// TIA Portal V17 export
// export: Created 2025-07-01T14:25:48.2523347Z, ExportSetting WithDefaults, DisplayName Totally Integrated Automation Portal, DisplayVersion V17 Update 8, DisplayName TIA Portal Openness, DisplayVersion V17 Update 8, DisplayName TIA Portal Version Control Interface, DisplayVersion V17, DisplayName SINAMICS Startdrive Advanced, DisplayVersion V17 SP2, DisplayName SINAMICS Startdrive G110M, G120, G120C, G120D, G120P, G115D, DisplayVersion V17 SP2, DisplayName SINAMICS Startdrive G130, G150, S120, S150, SINAMICS MV, S210, DisplayVersion V17 SP2, DisplayName STEP 7 Professional, DisplayVersion V17 Update 8, DisplayName SINUMERIK ONE STEP 7 Toolbox, DisplayVersion V17 Update 12, DisplayName SINUMERIK ONE PLC Basic Program Plus, DisplayVersion V17 Update 12, DisplayName SINUMERIK 840D sl STEP 7 Toolbox, DisplayVersion V17 Update 12, DisplayName STEP 7 Safety, DisplayVersion V17 Update 6, DisplayName WinCC Advanced, DisplayVersion V17 Update 8
FUNCTION "FC2103_ELECTRICAL_CABINET" : Void   // FC2103, LAD
{ S7_Optimized_Access := 'FALSE' }
AUTHOR : ETXETAR
VERSION : 1.0
// stored: AutoNumber false, IsIECCheckEnabled false, SetENOAutomatically false, UDAEnableTagReadback false
   VAR_TEMP
      PSP_ALARM_AUX : Bool;
   END_VAR
   VAR CONSTANT
      FC_NUMBER : DInt := 2103;
   END_VAR
   VAR_TEMP   // added for the SCL form of the ladder/FBD networks
      _w1 : Bool;
   END_VAR
BEGIN

REGION Network 1: INPUTS
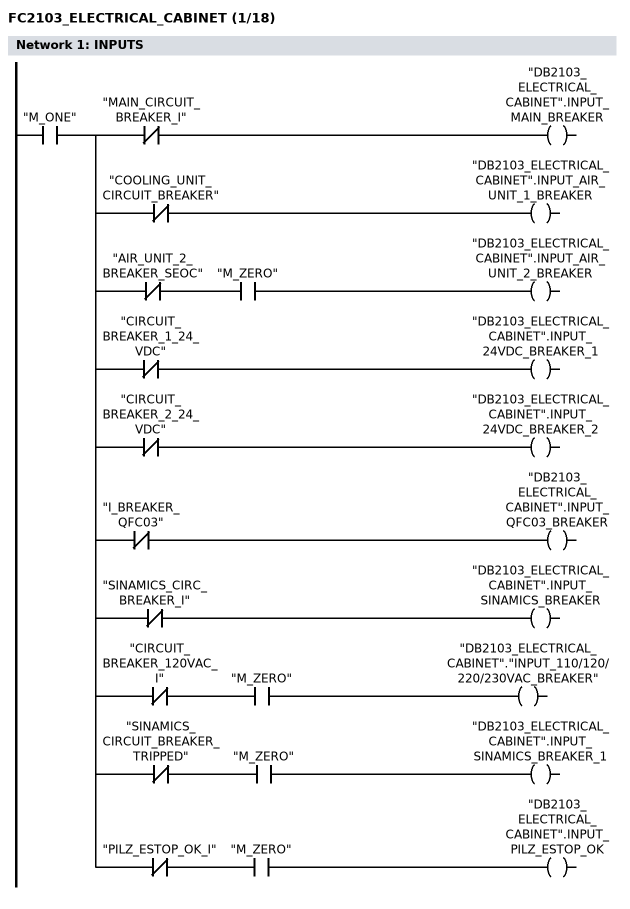
   RUNG wire#powerrail
      Contact( "M_ONE" )
      wire#w1
      I_Contact( "MAIN_CIRCUIT_BREAKER_I" )
      Coil( "DB2103_ELECTRICAL_CABINET".INPUT_MAIN_BREAKER )
   END_RUNG
   RUNG wire#w1
      I_Contact( "COOLING_UNIT_CIRCUIT_BREAKER" )
      Coil( "DB2103_ELECTRICAL_CABINET".INPUT_AIR_UNIT_1_BREAKER )
   END_RUNG
   RUNG wire#w1
      I_Contact( "AIR_UNIT_2_BREAKER_SEOC" )
      Contact( "M_ZERO" )
      Coil( "DB2103_ELECTRICAL_CABINET".INPUT_AIR_UNIT_2_BREAKER )
   END_RUNG
   RUNG wire#w1
      I_Contact( "CIRCUIT_BREAKER_1_24_VDC" )
      Coil( "DB2103_ELECTRICAL_CABINET".INPUT_24VDC_BREAKER_1 )
   END_RUNG
   RUNG wire#w1
      I_Contact( "CIRCUIT_BREAKER_2_24_VDC" )
      Coil( "DB2103_ELECTRICAL_CABINET".INPUT_24VDC_BREAKER_2 )
   END_RUNG
   RUNG wire#w1
      I_Contact( "I_BREAKER_QFC03" )
      Coil( "DB2103_ELECTRICAL_CABINET".INPUT_QFC03_BREAKER )
   END_RUNG
   RUNG wire#w1
      I_Contact( "SINAMICS_CIRC_BREAKER_I" )
      Coil( "DB2103_ELECTRICAL_CABINET".INPUT_SINAMICS_BREAKER )
   END_RUNG
   RUNG wire#w1
      I_Contact( "CIRCUIT_BREAKER_120VAC_I" )
      Contact( "M_ZERO" )
      Coil( "DB2103_ELECTRICAL_CABINET"."INPUT_110/120/220/230VAC_BREAKER" )
   END_RUNG
   RUNG wire#w1
      I_Contact( "SINAMICS_CIRCUIT_BREAKER_TRIPPED" )
      Contact( "M_ZERO" )
      Coil( "DB2103_ELECTRICAL_CABINET".INPUT_SINAMICS_BREAKER_1 )
   END_RUNG
   RUNG wire#w1
      I_Contact( "PILZ_ESTOP_OK_I" )
      Contact( "M_ZERO" )
      Coil( "DB2103_ELECTRICAL_CABINET".INPUT_PILZ_ESTOP_OK )
   END_RUNG
   // the same network as SCL:
   "DB2103_ELECTRICAL_CABINET".INPUT_MAIN_BREAKER := "M_ONE" AND NOT "MAIN_CIRCUIT_BREAKER_I";
   "DB2103_ELECTRICAL_CABINET".INPUT_AIR_UNIT_1_BREAKER := "M_ONE" AND NOT "COOLING_UNIT_CIRCUIT_BREAKER";
   "DB2103_ELECTRICAL_CABINET".INPUT_AIR_UNIT_2_BREAKER := "M_ONE" AND NOT "AIR_UNIT_2_BREAKER_SEOC" AND "M_ZERO";
   "DB2103_ELECTRICAL_CABINET".INPUT_24VDC_BREAKER_1 := "M_ONE" AND NOT "CIRCUIT_BREAKER_1_24_VDC";
   "DB2103_ELECTRICAL_CABINET".INPUT_24VDC_BREAKER_2 := "M_ONE" AND NOT "CIRCUIT_BREAKER_2_24_VDC";
   "DB2103_ELECTRICAL_CABINET".INPUT_QFC03_BREAKER := "M_ONE" AND NOT "I_BREAKER_QFC03";
   "DB2103_ELECTRICAL_CABINET".INPUT_SINAMICS_BREAKER := "M_ONE" AND NOT "SINAMICS_CIRC_BREAKER_I";
   "DB2103_ELECTRICAL_CABINET"."INPUT_110/120/220/230VAC_BREAKER" := "M_ONE" AND NOT "CIRCUIT_BREAKER_120VAC_I" AND "M_ZERO";
   "DB2103_ELECTRICAL_CABINET".INPUT_SINAMICS_BREAKER_1 := "M_ONE" AND NOT "SINAMICS_CIRCUIT_BREAKER_TRIPPED" AND "M_ZERO";
   "DB2103_ELECTRICAL_CABINET".INPUT_PILZ_ESTOP_OK := "M_ONE" AND NOT "PILZ_ESTOP_OK_I" AND "M_ZERO";
END_REGION

REGION Network 2: INPUTS
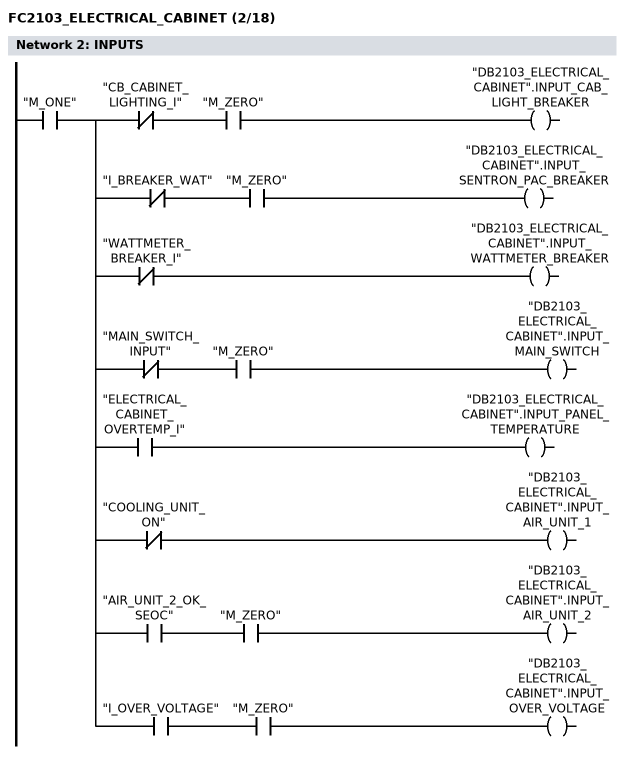
   RUNG wire#powerrail
      Contact( "M_ONE" )
      wire#w1
      I_Contact( "CB_CABINET_LIGHTING_I" )
      Contact( "M_ZERO" )
      Coil( "DB2103_ELECTRICAL_CABINET".INPUT_CAB_LIGHT_BREAKER )
   END_RUNG
   RUNG wire#w1
      I_Contact( "I_BREAKER_WAT" )
      Contact( "M_ZERO" )
      Coil( "DB2103_ELECTRICAL_CABINET".INPUT_SENTRON_PAC_BREAKER )
   END_RUNG
   RUNG wire#w1
      I_Contact( "WATTMETER_BREAKER_I" )
      Coil( "DB2103_ELECTRICAL_CABINET".INPUT_WATTMETER_BREAKER )
   END_RUNG
   RUNG wire#w1
      I_Contact( "MAIN_SWITCH_INPUT" )
      Contact( "M_ZERO" )
      Coil( "DB2103_ELECTRICAL_CABINET".INPUT_MAIN_SWITCH )
   END_RUNG
   RUNG wire#w1
      Contact( "ELECTRICAL_CABINET_OVERTEMP_I" )
      Coil( "DB2103_ELECTRICAL_CABINET".INPUT_PANEL_TEMPERATURE )
   END_RUNG
   RUNG wire#w1
      I_Contact( "COOLING_UNIT_ON" )
      Coil( "DB2103_ELECTRICAL_CABINET".INPUT_AIR_UNIT_1 )
   END_RUNG
   RUNG wire#w1
      Contact( "AIR_UNIT_2_OK_SEOC" )
      Contact( "M_ZERO" )
      Coil( "DB2103_ELECTRICAL_CABINET".INPUT_AIR_UNIT_2 )
   END_RUNG
   RUNG wire#w1
      Contact( "I_OVER_VOLTAGE" )
      Contact( "M_ZERO" )
      Coil( "DB2103_ELECTRICAL_CABINET".INPUT_OVER_VOLTAGE )
   END_RUNG
   // the same network as SCL:
   "DB2103_ELECTRICAL_CABINET".INPUT_CAB_LIGHT_BREAKER := "M_ONE" AND NOT "CB_CABINET_LIGHTING_I" AND "M_ZERO";
   "DB2103_ELECTRICAL_CABINET".INPUT_SENTRON_PAC_BREAKER := "M_ONE" AND NOT "I_BREAKER_WAT" AND "M_ZERO";
   "DB2103_ELECTRICAL_CABINET".INPUT_WATTMETER_BREAKER := "M_ONE" AND NOT "WATTMETER_BREAKER_I";
   "DB2103_ELECTRICAL_CABINET".INPUT_MAIN_SWITCH := "M_ONE" AND NOT "MAIN_SWITCH_INPUT" AND "M_ZERO";
   "DB2103_ELECTRICAL_CABINET".INPUT_PANEL_TEMPERATURE := "M_ONE" AND "ELECTRICAL_CABINET_OVERTEMP_I";
   "DB2103_ELECTRICAL_CABINET".INPUT_AIR_UNIT_1 := "M_ONE" AND NOT "COOLING_UNIT_ON";
   "DB2103_ELECTRICAL_CABINET".INPUT_AIR_UNIT_2 := "M_ONE" AND "AIR_UNIT_2_OK_SEOC" AND "M_ZERO";
   "DB2103_ELECTRICAL_CABINET".INPUT_OVER_VOLTAGE := "M_ONE" AND "I_OVER_VOLTAGE" AND "M_ZERO";
END_REGION

REGION Network 3: INPUTS
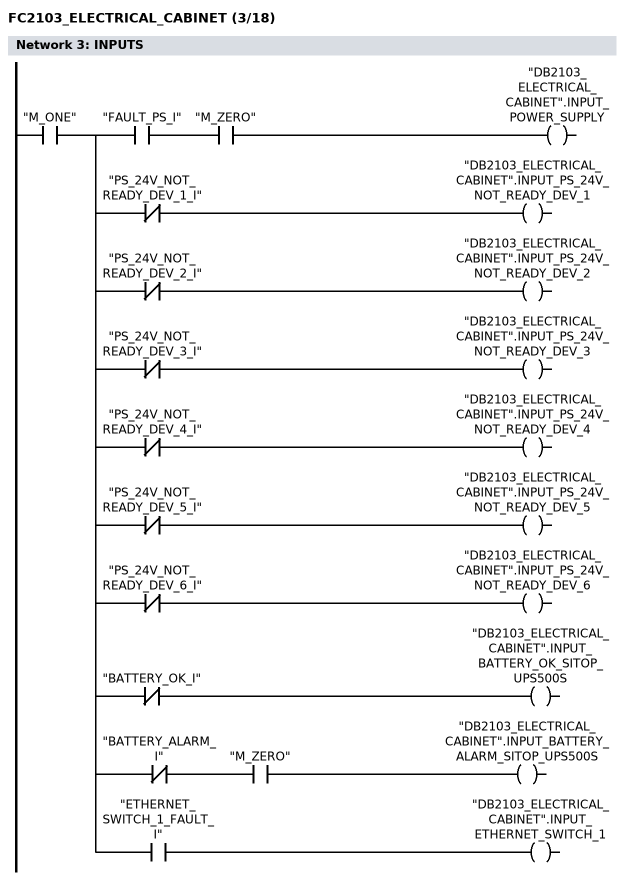
   RUNG wire#powerrail
      Contact( "M_ONE" )
      wire#w1
      Contact( "FAULT_PS_I" )
      Contact( "M_ZERO" )
      Coil( "DB2103_ELECTRICAL_CABINET".INPUT_POWER_SUPPLY )
   END_RUNG
   RUNG wire#w1
      I_Contact( "PS_24V_NOT_READY_DEV_1_I" )
      Coil( "DB2103_ELECTRICAL_CABINET".INPUT_PS_24V_NOT_READY_DEV_1 )
   END_RUNG
   RUNG wire#w1
      I_Contact( "PS_24V_NOT_READY_DEV_2_I" )
      Coil( "DB2103_ELECTRICAL_CABINET".INPUT_PS_24V_NOT_READY_DEV_2 )
   END_RUNG
   RUNG wire#w1
      I_Contact( "PS_24V_NOT_READY_DEV_3_I" )
      Coil( "DB2103_ELECTRICAL_CABINET".INPUT_PS_24V_NOT_READY_DEV_3 )
   END_RUNG
   RUNG wire#w1
      I_Contact( "PS_24V_NOT_READY_DEV_4_I" )
      Coil( "DB2103_ELECTRICAL_CABINET".INPUT_PS_24V_NOT_READY_DEV_4 )
   END_RUNG
   RUNG wire#w1
      I_Contact( "PS_24V_NOT_READY_DEV_5_I" )
      Coil( "DB2103_ELECTRICAL_CABINET".INPUT_PS_24V_NOT_READY_DEV_5 )
   END_RUNG
   RUNG wire#w1
      I_Contact( "PS_24V_NOT_READY_DEV_6_I" )
      Coil( "DB2103_ELECTRICAL_CABINET".INPUT_PS_24V_NOT_READY_DEV_6 )
   END_RUNG
   RUNG wire#w1
      I_Contact( "BATTERY_OK_I" )
      Coil( "DB2103_ELECTRICAL_CABINET".INPUT_BATTERY_OK_SITOP_UPS500S )
   END_RUNG
   RUNG wire#w1
      I_Contact( "BATTERY_ALARM_I" )
      Contact( "M_ZERO" )
      Coil( "DB2103_ELECTRICAL_CABINET".INPUT_BATTERY_ALARM_SITOP_UPS500S )
   END_RUNG
   RUNG wire#w1
      Contact( "ETHERNET_SWITCH_1_FAULT_I" )
      Coil( "DB2103_ELECTRICAL_CABINET".INPUT_ETHERNET_SWITCH_1 )
   END_RUNG
   // the same network as SCL:
   "DB2103_ELECTRICAL_CABINET".INPUT_POWER_SUPPLY := "M_ONE" AND "FAULT_PS_I" AND "M_ZERO";
   "DB2103_ELECTRICAL_CABINET".INPUT_PS_24V_NOT_READY_DEV_1 := "M_ONE" AND NOT "PS_24V_NOT_READY_DEV_1_I";
   "DB2103_ELECTRICAL_CABINET".INPUT_PS_24V_NOT_READY_DEV_2 := "M_ONE" AND NOT "PS_24V_NOT_READY_DEV_2_I";
   "DB2103_ELECTRICAL_CABINET".INPUT_PS_24V_NOT_READY_DEV_3 := "M_ONE" AND NOT "PS_24V_NOT_READY_DEV_3_I";
   "DB2103_ELECTRICAL_CABINET".INPUT_PS_24V_NOT_READY_DEV_4 := "M_ONE" AND NOT "PS_24V_NOT_READY_DEV_4_I";
   "DB2103_ELECTRICAL_CABINET".INPUT_PS_24V_NOT_READY_DEV_5 := "M_ONE" AND NOT "PS_24V_NOT_READY_DEV_5_I";
   "DB2103_ELECTRICAL_CABINET".INPUT_PS_24V_NOT_READY_DEV_6 := "M_ONE" AND NOT "PS_24V_NOT_READY_DEV_6_I";
   "DB2103_ELECTRICAL_CABINET".INPUT_BATTERY_OK_SITOP_UPS500S := "M_ONE" AND NOT "BATTERY_OK_I";
   "DB2103_ELECTRICAL_CABINET".INPUT_BATTERY_ALARM_SITOP_UPS500S := "M_ONE" AND NOT "BATTERY_ALARM_I" AND "M_ZERO";
   "DB2103_ELECTRICAL_CABINET".INPUT_ETHERNET_SWITCH_1 := "M_ONE" AND "ETHERNET_SWITCH_1_FAULT_I";
END_REGION

REGION Network 4: INPUTS
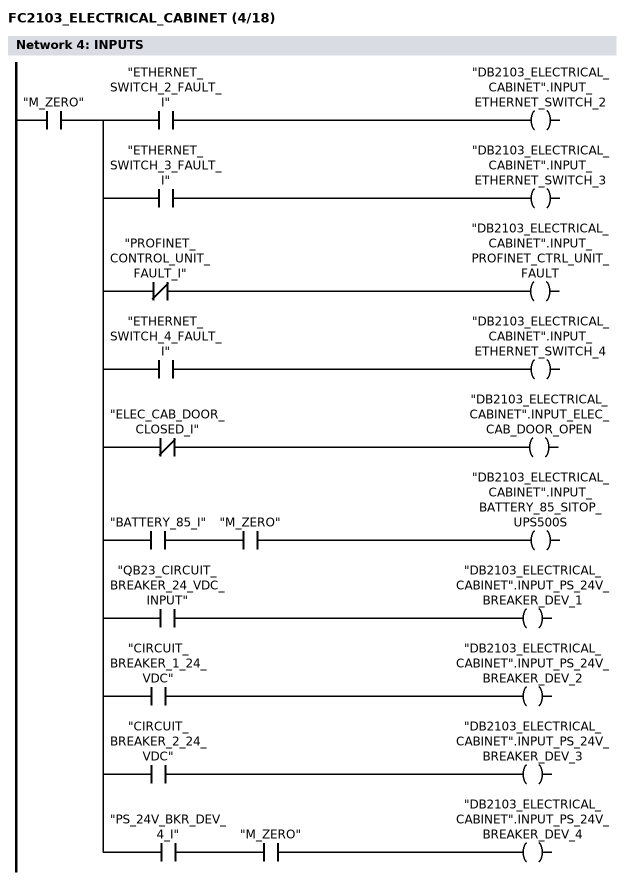
   RUNG wire#powerrail
      Contact( "M_ZERO" )
      wire#w1
      Contact( "ETHERNET_SWITCH_2_FAULT_I" )
      Coil( "DB2103_ELECTRICAL_CABINET".INPUT_ETHERNET_SWITCH_2 )
   END_RUNG
   RUNG wire#w1
      Contact( "ETHERNET_SWITCH_3_FAULT_I" )
      Coil( "DB2103_ELECTRICAL_CABINET".INPUT_ETHERNET_SWITCH_3 )
   END_RUNG
   RUNG wire#w1
      I_Contact( "PROFINET_CONTROL_UNIT_FAULT_I" )
      Coil( "DB2103_ELECTRICAL_CABINET".INPUT_PROFINET_CTRL_UNIT_FAULT )
   END_RUNG
   RUNG wire#w1
      Contact( "ETHERNET_SWITCH_4_FAULT_I" )
      Coil( "DB2103_ELECTRICAL_CABINET".INPUT_ETHERNET_SWITCH_4 )
   END_RUNG
   RUNG wire#w1
      I_Contact( "ELEC_CAB_DOOR_CLOSED_I" )
      Coil( "DB2103_ELECTRICAL_CABINET".INPUT_ELEC_CAB_DOOR_OPEN )
   END_RUNG
   RUNG wire#w1
      Contact( "BATTERY_85_I" )
      Contact( "M_ZERO" )
      Coil( "DB2103_ELECTRICAL_CABINET".INPUT_BATTERY_85_SITOP_UPS500S )
   END_RUNG
   RUNG wire#w1
      Contact( "QB23_CIRCUIT_BREAKER_24_VDC_INPUT" )
      Coil( "DB2103_ELECTRICAL_CABINET".INPUT_PS_24V_BREAKER_DEV_1 )
   END_RUNG
   RUNG wire#w1
      Contact( "CIRCUIT_BREAKER_1_24_VDC" )
      Coil( "DB2103_ELECTRICAL_CABINET".INPUT_PS_24V_BREAKER_DEV_2 )
   END_RUNG
   RUNG wire#w1
      Contact( "CIRCUIT_BREAKER_2_24_VDC" )
      Coil( "DB2103_ELECTRICAL_CABINET".INPUT_PS_24V_BREAKER_DEV_3 )
   END_RUNG
   RUNG wire#w1
      Contact( "PS_24V_BKR_DEV_4_I" )
      Contact( "M_ZERO" )
      Coil( "DB2103_ELECTRICAL_CABINET".INPUT_PS_24V_BREAKER_DEV_4 )
   END_RUNG
   // the same network as SCL:
   "DB2103_ELECTRICAL_CABINET".INPUT_ETHERNET_SWITCH_2 := "M_ZERO" AND "ETHERNET_SWITCH_2_FAULT_I";
   "DB2103_ELECTRICAL_CABINET".INPUT_ETHERNET_SWITCH_3 := "M_ZERO" AND "ETHERNET_SWITCH_3_FAULT_I";
   "DB2103_ELECTRICAL_CABINET".INPUT_PROFINET_CTRL_UNIT_FAULT := "M_ZERO" AND NOT "PROFINET_CONTROL_UNIT_FAULT_I";
   "DB2103_ELECTRICAL_CABINET".INPUT_ETHERNET_SWITCH_4 := "M_ZERO" AND "ETHERNET_SWITCH_4_FAULT_I";
   "DB2103_ELECTRICAL_CABINET".INPUT_ELEC_CAB_DOOR_OPEN := "M_ZERO" AND NOT "ELEC_CAB_DOOR_CLOSED_I";
   "DB2103_ELECTRICAL_CABINET".INPUT_BATTERY_85_SITOP_UPS500S := "M_ZERO" AND "BATTERY_85_I" AND "M_ZERO";
   "DB2103_ELECTRICAL_CABINET".INPUT_PS_24V_BREAKER_DEV_1 := "M_ZERO" AND "QB23_CIRCUIT_BREAKER_24_VDC_INPUT";
   "DB2103_ELECTRICAL_CABINET".INPUT_PS_24V_BREAKER_DEV_2 := "M_ZERO" AND "CIRCUIT_BREAKER_1_24_VDC";
   "DB2103_ELECTRICAL_CABINET".INPUT_PS_24V_BREAKER_DEV_3 := "M_ZERO" AND "CIRCUIT_BREAKER_2_24_VDC";
   "DB2103_ELECTRICAL_CABINET".INPUT_PS_24V_BREAKER_DEV_4 := "M_ZERO" AND "PS_24V_BKR_DEV_4_I" AND "M_ZERO";
END_REGION

REGION Network 5: INPUTS
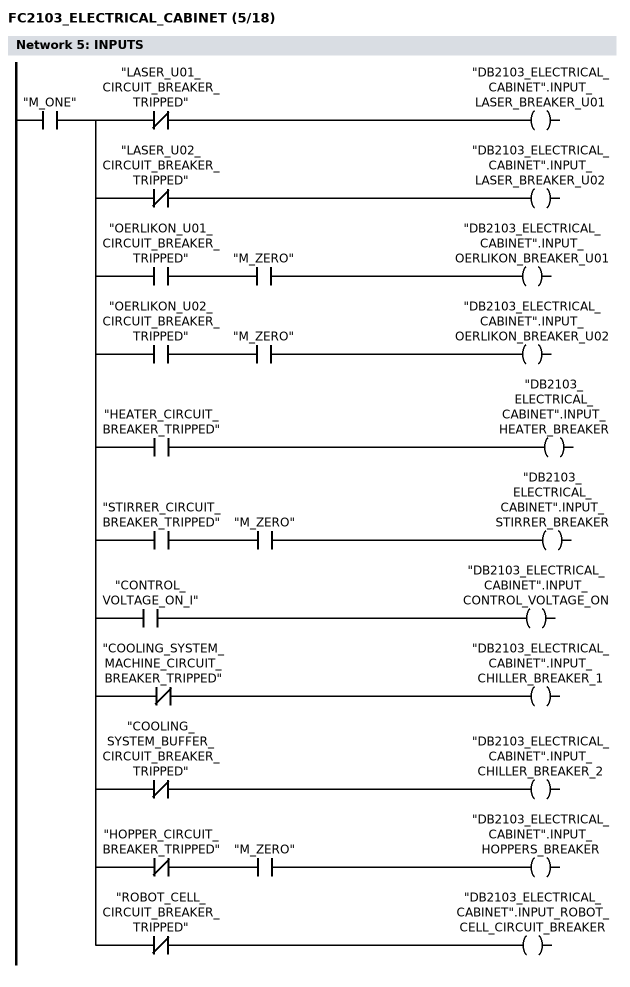
   RUNG wire#powerrail
      Contact( "M_ONE" )
      wire#w1
      I_Contact( "LASER_U01_CIRCUIT_BREAKER_TRIPPED" )
      Coil( "DB2103_ELECTRICAL_CABINET".INPUT_LASER_BREAKER_U01 )
   END_RUNG
   RUNG wire#w1
      I_Contact( "LASER_U02_CIRCUIT_BREAKER_TRIPPED" )
      Coil( "DB2103_ELECTRICAL_CABINET".INPUT_LASER_BREAKER_U02 )
   END_RUNG
   RUNG wire#w1
      Contact( "OERLIKON_U01_CIRCUIT_BREAKER_TRIPPED" )
      Contact( "M_ZERO" )
      Coil( "DB2103_ELECTRICAL_CABINET".INPUT_OERLIKON_BREAKER_U01 )
   END_RUNG
   RUNG wire#w1
      Contact( "OERLIKON_U02_CIRCUIT_BREAKER_TRIPPED" )
      Contact( "M_ZERO" )
      Coil( "DB2103_ELECTRICAL_CABINET".INPUT_OERLIKON_BREAKER_U02 )
   END_RUNG
   RUNG wire#w1
      Contact( "HEATER_CIRCUIT_BREAKER_TRIPPED" )
      Coil( "DB2103_ELECTRICAL_CABINET".INPUT_HEATER_BREAKER )
   END_RUNG
   RUNG wire#w1
      Contact( "STIRRER_CIRCUIT_BREAKER_TRIPPED" )
      Contact( "M_ZERO" )
      Coil( "DB2103_ELECTRICAL_CABINET".INPUT_STIRRER_BREAKER )
   END_RUNG
   RUNG wire#w1
      Contact( "CONTROL_VOLTAGE_ON_I" )
      Coil( "DB2103_ELECTRICAL_CABINET".INPUT_CONTROL_VOLTAGE_ON )
   END_RUNG
   RUNG wire#w1
      I_Contact( "COOLING_SYSTEM_MACHINE_CIRCUIT_BREAKER_TRIPPED" )
      Coil( "DB2103_ELECTRICAL_CABINET".INPUT_CHILLER_BREAKER_1 )
   END_RUNG
   RUNG wire#w1
      I_Contact( "COOLING_SYSTEM_BUFFER_CIRCUIT_BREAKER_TRIPPED" )
      Coil( "DB2103_ELECTRICAL_CABINET".INPUT_CHILLER_BREAKER_2 )
   END_RUNG
   RUNG wire#w1
      I_Contact( "HOPPER_CIRCUIT_BREAKER_TRIPPED" )
      Contact( "M_ZERO" )
      Coil( "DB2103_ELECTRICAL_CABINET".INPUT_HOPPERS_BREAKER )
   END_RUNG
   RUNG wire#w1
      I_Contact( "ROBOT_CELL_CIRCUIT_BREAKER_TRIPPED" )
      Coil( "DB2103_ELECTRICAL_CABINET".INPUT_ROBOT_CELL_CIRCUIT_BREAKER )
   END_RUNG
   // the same network as SCL:
   "DB2103_ELECTRICAL_CABINET".INPUT_LASER_BREAKER_U01 := "M_ONE" AND NOT "LASER_U01_CIRCUIT_BREAKER_TRIPPED";
   "DB2103_ELECTRICAL_CABINET".INPUT_LASER_BREAKER_U02 := "M_ONE" AND NOT "LASER_U02_CIRCUIT_BREAKER_TRIPPED";
   "DB2103_ELECTRICAL_CABINET".INPUT_OERLIKON_BREAKER_U01 := "M_ONE" AND "OERLIKON_U01_CIRCUIT_BREAKER_TRIPPED" AND "M_ZERO";
   "DB2103_ELECTRICAL_CABINET".INPUT_OERLIKON_BREAKER_U02 := "M_ONE" AND "OERLIKON_U02_CIRCUIT_BREAKER_TRIPPED" AND "M_ZERO";
   "DB2103_ELECTRICAL_CABINET".INPUT_HEATER_BREAKER := "M_ONE" AND "HEATER_CIRCUIT_BREAKER_TRIPPED";
   "DB2103_ELECTRICAL_CABINET".INPUT_STIRRER_BREAKER := "M_ONE" AND "STIRRER_CIRCUIT_BREAKER_TRIPPED" AND "M_ZERO";
   "DB2103_ELECTRICAL_CABINET".INPUT_CONTROL_VOLTAGE_ON := "M_ONE" AND "CONTROL_VOLTAGE_ON_I";
   "DB2103_ELECTRICAL_CABINET".INPUT_CHILLER_BREAKER_1 := "M_ONE" AND NOT "COOLING_SYSTEM_MACHINE_CIRCUIT_BREAKER_TRIPPED";
   "DB2103_ELECTRICAL_CABINET".INPUT_CHILLER_BREAKER_2 := "M_ONE" AND NOT "COOLING_SYSTEM_BUFFER_CIRCUIT_BREAKER_TRIPPED";
   "DB2103_ELECTRICAL_CABINET".INPUT_HOPPERS_BREAKER := "M_ONE" AND NOT "HOPPER_CIRCUIT_BREAKER_TRIPPED" AND "M_ZERO";
   "DB2103_ELECTRICAL_CABINET".INPUT_ROBOT_CELL_CIRCUIT_BREAKER := "M_ONE" AND NOT "ROBOT_CELL_CIRCUIT_BREAKER_TRIPPED";
END_REGION

REGION Network 6: INPUTS
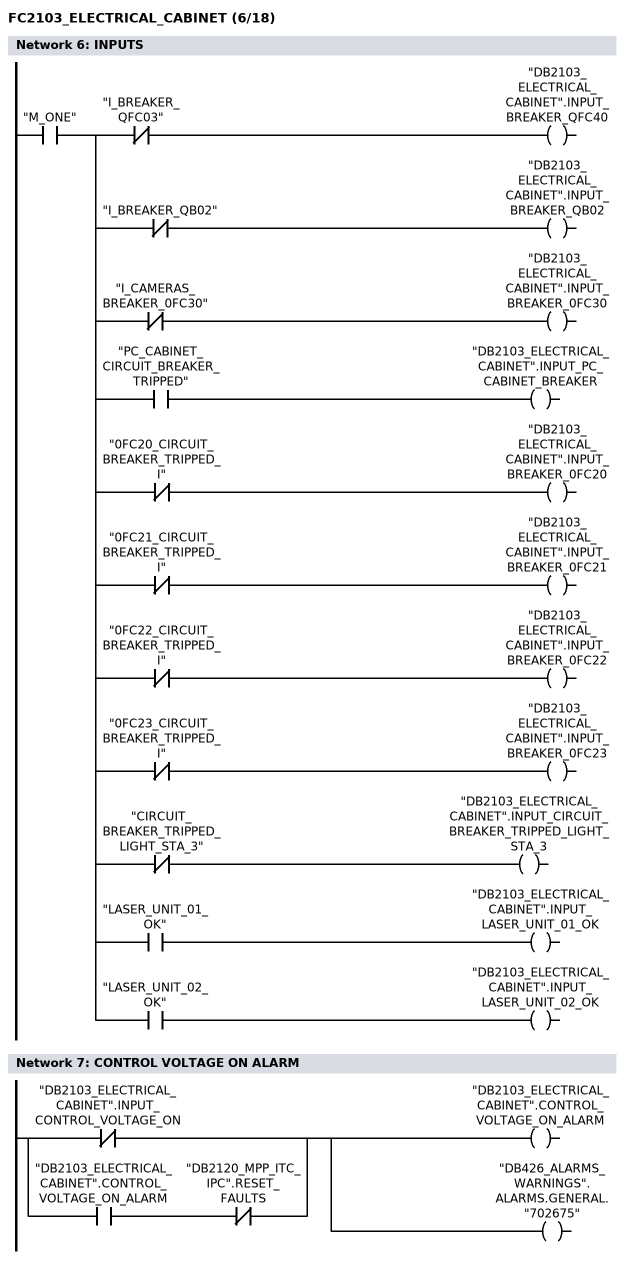
   RUNG wire#powerrail
      Contact( "M_ONE" )
      wire#w1
      I_Contact( "I_BREAKER_QFC03" )
      Coil( "DB2103_ELECTRICAL_CABINET".INPUT_BREAKER_QFC40 )
   END_RUNG
   RUNG wire#w1
      I_Contact( "I_BREAKER_QB02" )
      Coil( "DB2103_ELECTRICAL_CABINET".INPUT_BREAKER_QB02 )
   END_RUNG
   RUNG wire#w1
      I_Contact( "I_CAMERAS_BREAKER_0FC30" )
      Coil( "DB2103_ELECTRICAL_CABINET".INPUT_BREAKER_0FC30 )
   END_RUNG
   RUNG wire#w1
      Contact( "PC_CABINET_CIRCUIT_BREAKER_TRIPPED" )
      Coil( "DB2103_ELECTRICAL_CABINET".INPUT_PC_CABINET_BREAKER )
   END_RUNG
   RUNG wire#w1
      I_Contact( "0FC20_CIRCUIT_BREAKER_TRIPPED_I" )
      Coil( "DB2103_ELECTRICAL_CABINET".INPUT_BREAKER_0FC20 )
   END_RUNG
   RUNG wire#w1
      I_Contact( "0FC21_CIRCUIT_BREAKER_TRIPPED_I" )
      Coil( "DB2103_ELECTRICAL_CABINET".INPUT_BREAKER_0FC21 )
   END_RUNG
   RUNG wire#w1
      I_Contact( "0FC22_CIRCUIT_BREAKER_TRIPPED_I" )
      Coil( "DB2103_ELECTRICAL_CABINET".INPUT_BREAKER_0FC22 )
   END_RUNG
   RUNG wire#w1
      I_Contact( "0FC23_CIRCUIT_BREAKER_TRIPPED_I" )
      Coil( "DB2103_ELECTRICAL_CABINET".INPUT_BREAKER_0FC23 )
   END_RUNG
   RUNG wire#w1
      I_Contact( "CIRCUIT_BREAKER_TRIPPED_LIGHT_STA_3" )
      Coil( "DB2103_ELECTRICAL_CABINET".INPUT_CIRCUIT_BREAKER_TRIPPED_LIGHT_STA_3 )
   END_RUNG
   RUNG wire#w1
      Contact( "LASER_UNIT_01_OK" )
      Coil( "DB2103_ELECTRICAL_CABINET".INPUT_LASER_UNIT_01_OK )
   END_RUNG
   RUNG wire#w1
      Contact( "LASER_UNIT_02_OK" )
      Coil( "DB2103_ELECTRICAL_CABINET".INPUT_LASER_UNIT_02_OK )
   END_RUNG
   // the same network as SCL:
   "DB2103_ELECTRICAL_CABINET".INPUT_BREAKER_QFC40 := "M_ONE" AND NOT "I_BREAKER_QFC03";
   "DB2103_ELECTRICAL_CABINET".INPUT_BREAKER_QB02 := "M_ONE" AND NOT "I_BREAKER_QB02";
   "DB2103_ELECTRICAL_CABINET".INPUT_BREAKER_0FC30 := "M_ONE" AND NOT "I_CAMERAS_BREAKER_0FC30";
   "DB2103_ELECTRICAL_CABINET".INPUT_PC_CABINET_BREAKER := "M_ONE" AND "PC_CABINET_CIRCUIT_BREAKER_TRIPPED";
   "DB2103_ELECTRICAL_CABINET".INPUT_BREAKER_0FC20 := "M_ONE" AND NOT "0FC20_CIRCUIT_BREAKER_TRIPPED_I";
   "DB2103_ELECTRICAL_CABINET".INPUT_BREAKER_0FC21 := "M_ONE" AND NOT "0FC21_CIRCUIT_BREAKER_TRIPPED_I";
   "DB2103_ELECTRICAL_CABINET".INPUT_BREAKER_0FC22 := "M_ONE" AND NOT "0FC22_CIRCUIT_BREAKER_TRIPPED_I";
   "DB2103_ELECTRICAL_CABINET".INPUT_BREAKER_0FC23 := "M_ONE" AND NOT "0FC23_CIRCUIT_BREAKER_TRIPPED_I";
   "DB2103_ELECTRICAL_CABINET".INPUT_CIRCUIT_BREAKER_TRIPPED_LIGHT_STA_3 := "M_ONE" AND NOT "CIRCUIT_BREAKER_TRIPPED_LIGHT_STA_3";
   "DB2103_ELECTRICAL_CABINET".INPUT_LASER_UNIT_01_OK := "M_ONE" AND "LASER_UNIT_01_OK";
   "DB2103_ELECTRICAL_CABINET".INPUT_LASER_UNIT_02_OK := "M_ONE" AND "LASER_UNIT_02_OK";
END_REGION

REGION Network 7: CONTROL VOLTAGE ON ALARM
   RUNG wire#powerrail
      I_Contact( "DB2103_ELECTRICAL_CABINET".INPUT_CONTROL_VOLTAGE_ON )
      wire#w1
      Coil( "DB2103_ELECTRICAL_CABINET".CONTROL_VOLTAGE_ON_ALARM )
   END_RUNG
   RUNG wire#powerrail
      Contact( "DB2103_ELECTRICAL_CABINET".CONTROL_VOLTAGE_ON_ALARM )
      I_Contact( "DB2120_MPP_ITC_IPC".RESET_FAULTS )
   END_RUNG wire#w1
   RUNG wire#w1
      Coil( "DB426_ALARMS_WARNINGS".ALARMS.GENERAL."702675" )
   END_RUNG
   // the same network as SCL:
   "DB2103_ELECTRICAL_CABINET".CONTROL_VOLTAGE_ON_ALARM := NOT "DB2103_ELECTRICAL_CABINET".INPUT_CONTROL_VOLTAGE_ON OR ("DB2103_ELECTRICAL_CABINET".CONTROL_VOLTAGE_ON_ALARM AND NOT "DB2120_MPP_ITC_IPC".RESET_FAULTS);
   "DB426_ALARMS_WARNINGS".ALARMS.GENERAL."702675" := "DB2103_ELECTRICAL_CABINET".CONTROL_VOLTAGE_ON_ALARM;
END_REGION

REGION Network 8: MAIN CIRCUIT BREAKER TRIPPED ALARM
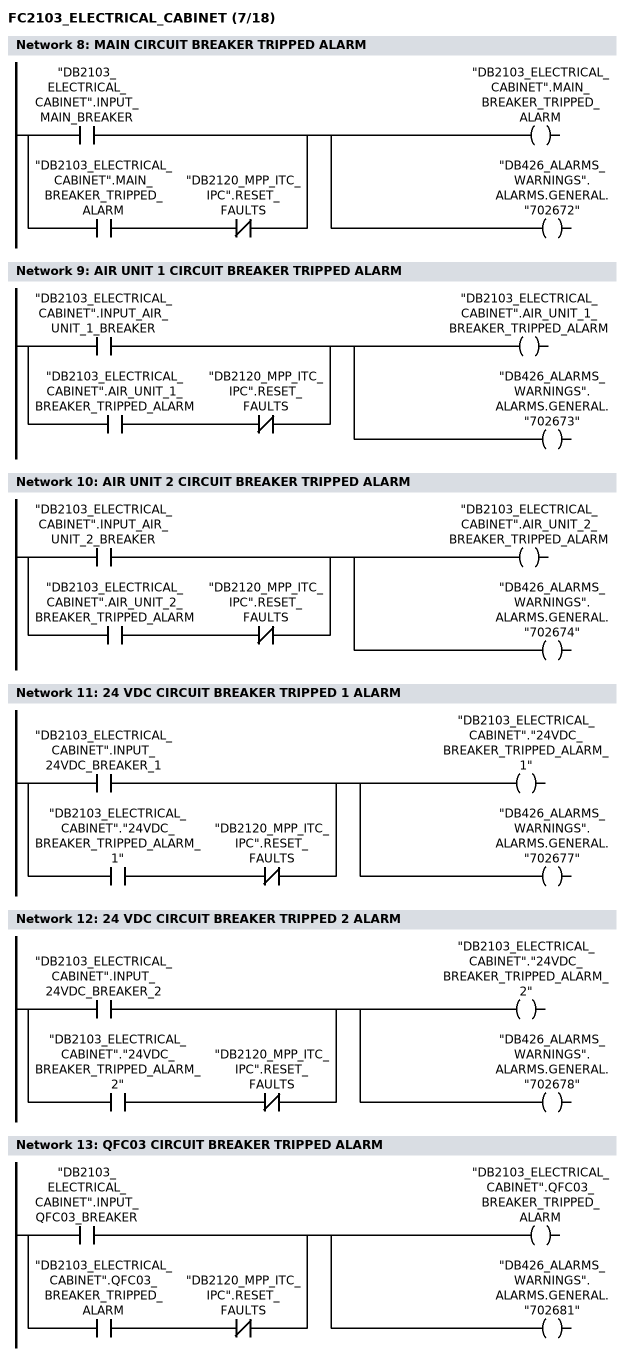
   RUNG wire#powerrail
      Contact( "DB2103_ELECTRICAL_CABINET".INPUT_MAIN_BREAKER )
      wire#w1
      Coil( "DB2103_ELECTRICAL_CABINET".MAIN_BREAKER_TRIPPED_ALARM )
   END_RUNG
   RUNG wire#powerrail
      Contact( "DB2103_ELECTRICAL_CABINET".MAIN_BREAKER_TRIPPED_ALARM )
      I_Contact( "DB2120_MPP_ITC_IPC".RESET_FAULTS )
   END_RUNG wire#w1
   RUNG wire#w1
      Coil( "DB426_ALARMS_WARNINGS".ALARMS.GENERAL."702672" )
   END_RUNG
   // the same network as SCL:
   "DB2103_ELECTRICAL_CABINET".MAIN_BREAKER_TRIPPED_ALARM := "DB2103_ELECTRICAL_CABINET".INPUT_MAIN_BREAKER OR ("DB2103_ELECTRICAL_CABINET".MAIN_BREAKER_TRIPPED_ALARM AND NOT "DB2120_MPP_ITC_IPC".RESET_FAULTS);
   "DB426_ALARMS_WARNINGS".ALARMS.GENERAL."702672" := "DB2103_ELECTRICAL_CABINET".MAIN_BREAKER_TRIPPED_ALARM;
END_REGION

REGION Network 9: AIR UNIT 1 CIRCUIT BREAKER TRIPPED ALARM
   RUNG wire#powerrail
      Contact( "DB2103_ELECTRICAL_CABINET".INPUT_AIR_UNIT_1_BREAKER )
      wire#w1
      Coil( "DB2103_ELECTRICAL_CABINET".AIR_UNIT_1_BREAKER_TRIPPED_ALARM )
   END_RUNG
   RUNG wire#powerrail
      Contact( "DB2103_ELECTRICAL_CABINET".AIR_UNIT_1_BREAKER_TRIPPED_ALARM )
      I_Contact( "DB2120_MPP_ITC_IPC".RESET_FAULTS )
   END_RUNG wire#w1
   RUNG wire#w1
      Coil( "DB426_ALARMS_WARNINGS".ALARMS.GENERAL."702673" )
   END_RUNG
   // the same network as SCL:
   "DB2103_ELECTRICAL_CABINET".AIR_UNIT_1_BREAKER_TRIPPED_ALARM := "DB2103_ELECTRICAL_CABINET".INPUT_AIR_UNIT_1_BREAKER OR ("DB2103_ELECTRICAL_CABINET".AIR_UNIT_1_BREAKER_TRIPPED_ALARM AND NOT "DB2120_MPP_ITC_IPC".RESET_FAULTS);
   "DB426_ALARMS_WARNINGS".ALARMS.GENERAL."702673" := "DB2103_ELECTRICAL_CABINET".AIR_UNIT_1_BREAKER_TRIPPED_ALARM;
END_REGION

REGION Network 10: AIR UNIT 2 CIRCUIT BREAKER TRIPPED ALARM
   RUNG wire#powerrail
      Contact( "DB2103_ELECTRICAL_CABINET".INPUT_AIR_UNIT_2_BREAKER )
      wire#w1
      Coil( "DB2103_ELECTRICAL_CABINET".AIR_UNIT_2_BREAKER_TRIPPED_ALARM )
   END_RUNG
   RUNG wire#powerrail
      Contact( "DB2103_ELECTRICAL_CABINET".AIR_UNIT_2_BREAKER_TRIPPED_ALARM )
      I_Contact( "DB2120_MPP_ITC_IPC".RESET_FAULTS )
   END_RUNG wire#w1
   RUNG wire#w1
      Coil( "DB426_ALARMS_WARNINGS".ALARMS.GENERAL."702674" )
   END_RUNG
   // the same network as SCL:
   "DB2103_ELECTRICAL_CABINET".AIR_UNIT_2_BREAKER_TRIPPED_ALARM := "DB2103_ELECTRICAL_CABINET".INPUT_AIR_UNIT_2_BREAKER OR ("DB2103_ELECTRICAL_CABINET".AIR_UNIT_2_BREAKER_TRIPPED_ALARM AND NOT "DB2120_MPP_ITC_IPC".RESET_FAULTS);
   "DB426_ALARMS_WARNINGS".ALARMS.GENERAL."702674" := "DB2103_ELECTRICAL_CABINET".AIR_UNIT_2_BREAKER_TRIPPED_ALARM;
END_REGION

REGION Network 11: 24 VDC CIRCUIT BREAKER TRIPPED 1 ALARM
   RUNG wire#powerrail
      Contact( "DB2103_ELECTRICAL_CABINET".INPUT_24VDC_BREAKER_1 )
      wire#w1
      Coil( "DB2103_ELECTRICAL_CABINET"."24VDC_BREAKER_TRIPPED_ALARM_1" )
   END_RUNG
   RUNG wire#powerrail
      Contact( "DB2103_ELECTRICAL_CABINET"."24VDC_BREAKER_TRIPPED_ALARM_1" )
      I_Contact( "DB2120_MPP_ITC_IPC".RESET_FAULTS )
   END_RUNG wire#w1
   RUNG wire#w1
      Coil( "DB426_ALARMS_WARNINGS".ALARMS.GENERAL."702677" )
   END_RUNG
   // the same network as SCL:
   "DB2103_ELECTRICAL_CABINET"."24VDC_BREAKER_TRIPPED_ALARM_1" := "DB2103_ELECTRICAL_CABINET".INPUT_24VDC_BREAKER_1 OR ("DB2103_ELECTRICAL_CABINET"."24VDC_BREAKER_TRIPPED_ALARM_1" AND NOT "DB2120_MPP_ITC_IPC".RESET_FAULTS);
   "DB426_ALARMS_WARNINGS".ALARMS.GENERAL."702677" := "DB2103_ELECTRICAL_CABINET"."24VDC_BREAKER_TRIPPED_ALARM_1";
END_REGION

REGION Network 12: 24 VDC CIRCUIT BREAKER TRIPPED 2 ALARM
   RUNG wire#powerrail
      Contact( "DB2103_ELECTRICAL_CABINET".INPUT_24VDC_BREAKER_2 )
      wire#w1
      Coil( "DB2103_ELECTRICAL_CABINET"."24VDC_BREAKER_TRIPPED_ALARM_2" )
   END_RUNG
   RUNG wire#powerrail
      Contact( "DB2103_ELECTRICAL_CABINET"."24VDC_BREAKER_TRIPPED_ALARM_2" )
      I_Contact( "DB2120_MPP_ITC_IPC".RESET_FAULTS )
   END_RUNG wire#w1
   RUNG wire#w1
      Coil( "DB426_ALARMS_WARNINGS".ALARMS.GENERAL."702678" )
   END_RUNG
   // the same network as SCL:
   "DB2103_ELECTRICAL_CABINET"."24VDC_BREAKER_TRIPPED_ALARM_2" := "DB2103_ELECTRICAL_CABINET".INPUT_24VDC_BREAKER_2 OR ("DB2103_ELECTRICAL_CABINET"."24VDC_BREAKER_TRIPPED_ALARM_2" AND NOT "DB2120_MPP_ITC_IPC".RESET_FAULTS);
   "DB426_ALARMS_WARNINGS".ALARMS.GENERAL."702678" := "DB2103_ELECTRICAL_CABINET"."24VDC_BREAKER_TRIPPED_ALARM_2";
END_REGION

REGION Network 13: QFC03 CIRCUIT BREAKER TRIPPED ALARM
   RUNG wire#powerrail
      Contact( "DB2103_ELECTRICAL_CABINET".INPUT_QFC03_BREAKER )
      wire#w1
      Coil( "DB2103_ELECTRICAL_CABINET".QFC03_BREAKER_TRIPPED_ALARM )
   END_RUNG
   RUNG wire#powerrail
      Contact( "DB2103_ELECTRICAL_CABINET".QFC03_BREAKER_TRIPPED_ALARM )
      I_Contact( "DB2120_MPP_ITC_IPC".RESET_FAULTS )
   END_RUNG wire#w1
   RUNG wire#w1
      Coil( "DB426_ALARMS_WARNINGS".ALARMS.GENERAL."702681" )
   END_RUNG
   // the same network as SCL:
   "DB2103_ELECTRICAL_CABINET".QFC03_BREAKER_TRIPPED_ALARM := "DB2103_ELECTRICAL_CABINET".INPUT_QFC03_BREAKER OR ("DB2103_ELECTRICAL_CABINET".QFC03_BREAKER_TRIPPED_ALARM AND NOT "DB2120_MPP_ITC_IPC".RESET_FAULTS);
   "DB426_ALARMS_WARNINGS".ALARMS.GENERAL."702681" := "DB2103_ELECTRICAL_CABINET".QFC03_BREAKER_TRIPPED_ALARM;
END_REGION

REGION Network 14: SINAMICS CIRCUIT BREAKER TRIPPED ALARM
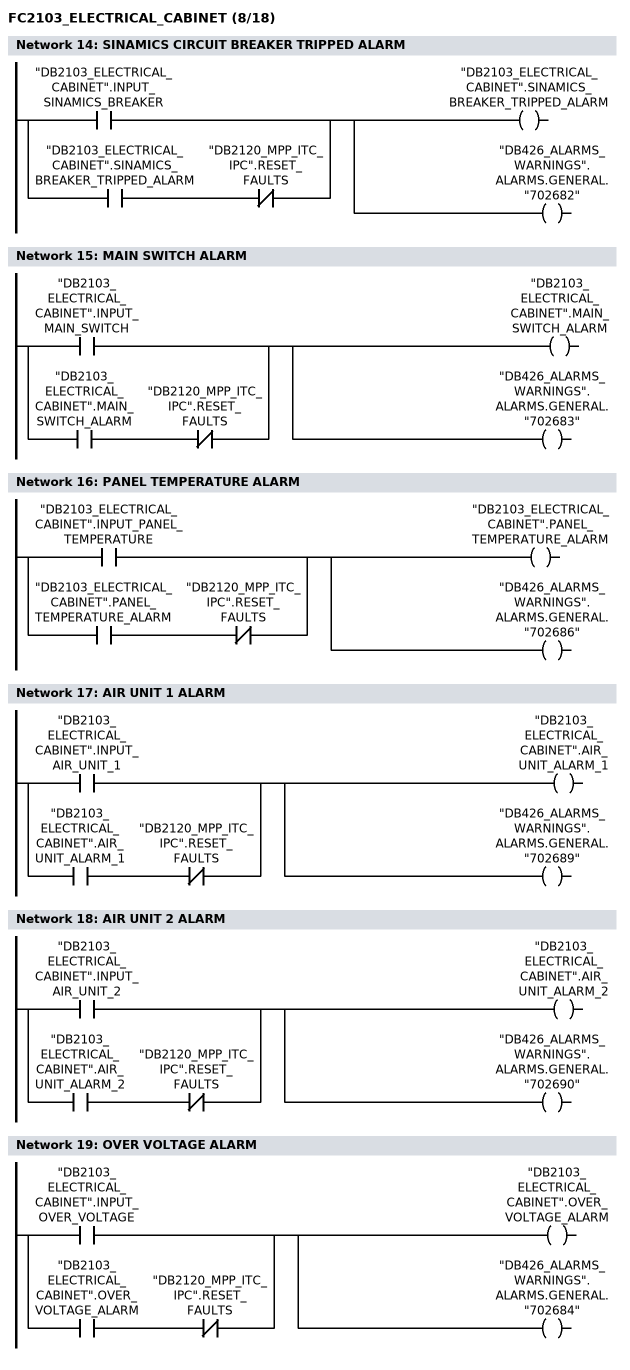
   RUNG wire#powerrail
      Contact( "DB2103_ELECTRICAL_CABINET".INPUT_SINAMICS_BREAKER )
      wire#w1
      Coil( "DB2103_ELECTRICAL_CABINET".SINAMICS_BREAKER_TRIPPED_ALARM )
   END_RUNG
   RUNG wire#powerrail
      Contact( "DB2103_ELECTRICAL_CABINET".SINAMICS_BREAKER_TRIPPED_ALARM )
      I_Contact( "DB2120_MPP_ITC_IPC".RESET_FAULTS )
   END_RUNG wire#w1
   RUNG wire#w1
      Coil( "DB426_ALARMS_WARNINGS".ALARMS.GENERAL."702682" )
   END_RUNG
   // the same network as SCL:
   "DB2103_ELECTRICAL_CABINET".SINAMICS_BREAKER_TRIPPED_ALARM := "DB2103_ELECTRICAL_CABINET".INPUT_SINAMICS_BREAKER OR ("DB2103_ELECTRICAL_CABINET".SINAMICS_BREAKER_TRIPPED_ALARM AND NOT "DB2120_MPP_ITC_IPC".RESET_FAULTS);
   "DB426_ALARMS_WARNINGS".ALARMS.GENERAL."702682" := "DB2103_ELECTRICAL_CABINET".SINAMICS_BREAKER_TRIPPED_ALARM;
END_REGION

REGION Network 15: MAIN SWITCH ALARM
   RUNG wire#powerrail
      Contact( "DB2103_ELECTRICAL_CABINET".INPUT_MAIN_SWITCH )
      wire#w1
      Coil( "DB2103_ELECTRICAL_CABINET".MAIN_SWITCH_ALARM )
   END_RUNG
   RUNG wire#powerrail
      Contact( "DB2103_ELECTRICAL_CABINET".MAIN_SWITCH_ALARM )
      I_Contact( "DB2120_MPP_ITC_IPC".RESET_FAULTS )
   END_RUNG wire#w1
   RUNG wire#w1
      Coil( "DB426_ALARMS_WARNINGS".ALARMS.GENERAL."702683" )
   END_RUNG
   // the same network as SCL:
   "DB2103_ELECTRICAL_CABINET".MAIN_SWITCH_ALARM := "DB2103_ELECTRICAL_CABINET".INPUT_MAIN_SWITCH OR ("DB2103_ELECTRICAL_CABINET".MAIN_SWITCH_ALARM AND NOT "DB2120_MPP_ITC_IPC".RESET_FAULTS);
   "DB426_ALARMS_WARNINGS".ALARMS.GENERAL."702683" := "DB2103_ELECTRICAL_CABINET".MAIN_SWITCH_ALARM;
END_REGION

REGION Network 16: PANEL TEMPERATURE ALARM
   RUNG wire#powerrail
      Contact( "DB2103_ELECTRICAL_CABINET".INPUT_PANEL_TEMPERATURE )
      wire#w1
      Coil( "DB2103_ELECTRICAL_CABINET".PANEL_TEMPERATURE_ALARM )
   END_RUNG
   RUNG wire#powerrail
      Contact( "DB2103_ELECTRICAL_CABINET".PANEL_TEMPERATURE_ALARM )
      I_Contact( "DB2120_MPP_ITC_IPC".RESET_FAULTS )
   END_RUNG wire#w1
   RUNG wire#w1
      Coil( "DB426_ALARMS_WARNINGS".ALARMS.GENERAL."702686" )
   END_RUNG
   // the same network as SCL:
   "DB2103_ELECTRICAL_CABINET".PANEL_TEMPERATURE_ALARM := "DB2103_ELECTRICAL_CABINET".INPUT_PANEL_TEMPERATURE OR ("DB2103_ELECTRICAL_CABINET".PANEL_TEMPERATURE_ALARM AND NOT "DB2120_MPP_ITC_IPC".RESET_FAULTS);
   "DB426_ALARMS_WARNINGS".ALARMS.GENERAL."702686" := "DB2103_ELECTRICAL_CABINET".PANEL_TEMPERATURE_ALARM;
END_REGION

REGION Network 17: AIR UNIT 1 ALARM
   RUNG wire#powerrail
      Contact( "DB2103_ELECTRICAL_CABINET".INPUT_AIR_UNIT_1 )
      wire#w1
      Coil( "DB2103_ELECTRICAL_CABINET".AIR_UNIT_ALARM_1 )
   END_RUNG
   RUNG wire#powerrail
      Contact( "DB2103_ELECTRICAL_CABINET".AIR_UNIT_ALARM_1 )
      I_Contact( "DB2120_MPP_ITC_IPC".RESET_FAULTS )
   END_RUNG wire#w1
   RUNG wire#w1
      Coil( "DB426_ALARMS_WARNINGS".ALARMS.GENERAL."702689" )
   END_RUNG
   // the same network as SCL:
   "DB2103_ELECTRICAL_CABINET".AIR_UNIT_ALARM_1 := "DB2103_ELECTRICAL_CABINET".INPUT_AIR_UNIT_1 OR ("DB2103_ELECTRICAL_CABINET".AIR_UNIT_ALARM_1 AND NOT "DB2120_MPP_ITC_IPC".RESET_FAULTS);
   "DB426_ALARMS_WARNINGS".ALARMS.GENERAL."702689" := "DB2103_ELECTRICAL_CABINET".AIR_UNIT_ALARM_1;
END_REGION

REGION Network 18: AIR UNIT 2 ALARM
   RUNG wire#powerrail
      Contact( "DB2103_ELECTRICAL_CABINET".INPUT_AIR_UNIT_2 )
      wire#w1
      Coil( "DB2103_ELECTRICAL_CABINET".AIR_UNIT_ALARM_2 )
   END_RUNG
   RUNG wire#powerrail
      Contact( "DB2103_ELECTRICAL_CABINET".AIR_UNIT_ALARM_2 )
      I_Contact( "DB2120_MPP_ITC_IPC".RESET_FAULTS )
   END_RUNG wire#w1
   RUNG wire#w1
      Coil( "DB426_ALARMS_WARNINGS".ALARMS.GENERAL."702690" )
   END_RUNG
   // the same network as SCL:
   "DB2103_ELECTRICAL_CABINET".AIR_UNIT_ALARM_2 := "DB2103_ELECTRICAL_CABINET".INPUT_AIR_UNIT_2 OR ("DB2103_ELECTRICAL_CABINET".AIR_UNIT_ALARM_2 AND NOT "DB2120_MPP_ITC_IPC".RESET_FAULTS);
   "DB426_ALARMS_WARNINGS".ALARMS.GENERAL."702690" := "DB2103_ELECTRICAL_CABINET".AIR_UNIT_ALARM_2;
END_REGION

REGION Network 19: OVER VOLTAGE ALARM
   RUNG wire#powerrail
      Contact( "DB2103_ELECTRICAL_CABINET".INPUT_OVER_VOLTAGE )
      wire#w1
      Coil( "DB2103_ELECTRICAL_CABINET".OVER_VOLTAGE_ALARM )
   END_RUNG
   RUNG wire#powerrail
      Contact( "DB2103_ELECTRICAL_CABINET".OVER_VOLTAGE_ALARM )
      I_Contact( "DB2120_MPP_ITC_IPC".RESET_FAULTS )
   END_RUNG wire#w1
   RUNG wire#w1
      Coil( "DB426_ALARMS_WARNINGS".ALARMS.GENERAL."702684" )
   END_RUNG
   // the same network as SCL:
   "DB2103_ELECTRICAL_CABINET".OVER_VOLTAGE_ALARM := "DB2103_ELECTRICAL_CABINET".INPUT_OVER_VOLTAGE OR ("DB2103_ELECTRICAL_CABINET".OVER_VOLTAGE_ALARM AND NOT "DB2120_MPP_ITC_IPC".RESET_FAULTS);
   "DB426_ALARMS_WARNINGS".ALARMS.GENERAL."702684" := "DB2103_ELECTRICAL_CABINET".OVER_VOLTAGE_ALARM;
END_REGION

REGION Network 20: POWER SUPPLY ALARM
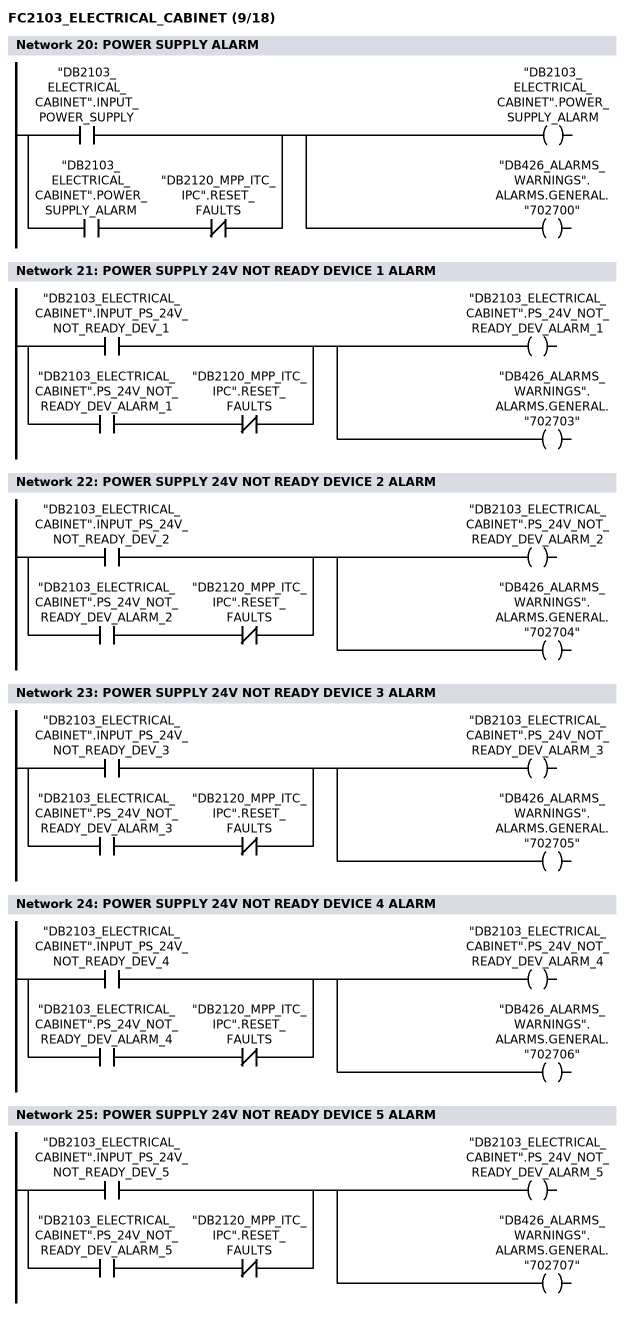
   RUNG wire#powerrail
      Contact( "DB2103_ELECTRICAL_CABINET".INPUT_POWER_SUPPLY )
      wire#w1
      Coil( "DB2103_ELECTRICAL_CABINET".POWER_SUPPLY_ALARM )
   END_RUNG
   RUNG wire#powerrail
      Contact( "DB2103_ELECTRICAL_CABINET".POWER_SUPPLY_ALARM )
      I_Contact( "DB2120_MPP_ITC_IPC".RESET_FAULTS )
   END_RUNG wire#w1
   RUNG wire#w1
      Coil( "DB426_ALARMS_WARNINGS".ALARMS.GENERAL."702700" )
   END_RUNG
   // the same network as SCL:
   "DB2103_ELECTRICAL_CABINET".POWER_SUPPLY_ALARM := "DB2103_ELECTRICAL_CABINET".INPUT_POWER_SUPPLY OR ("DB2103_ELECTRICAL_CABINET".POWER_SUPPLY_ALARM AND NOT "DB2120_MPP_ITC_IPC".RESET_FAULTS);
   "DB426_ALARMS_WARNINGS".ALARMS.GENERAL."702700" := "DB2103_ELECTRICAL_CABINET".POWER_SUPPLY_ALARM;
END_REGION

REGION Network 21: POWER SUPPLY 24V NOT READY DEVICE 1 ALARM
   RUNG wire#powerrail
      Contact( "DB2103_ELECTRICAL_CABINET".INPUT_PS_24V_NOT_READY_DEV_1 )
      wire#w1
      Coil( "DB2103_ELECTRICAL_CABINET".PS_24V_NOT_READY_DEV_ALARM_1 )
   END_RUNG
   RUNG wire#powerrail
      Contact( "DB2103_ELECTRICAL_CABINET".PS_24V_NOT_READY_DEV_ALARM_1 )
      I_Contact( "DB2120_MPP_ITC_IPC".RESET_FAULTS )
   END_RUNG wire#w1
   RUNG wire#w1
      Coil( "DB426_ALARMS_WARNINGS".ALARMS.GENERAL."702703" )
   END_RUNG
   // the same network as SCL:
   "DB2103_ELECTRICAL_CABINET".PS_24V_NOT_READY_DEV_ALARM_1 := "DB2103_ELECTRICAL_CABINET".INPUT_PS_24V_NOT_READY_DEV_1 OR ("DB2103_ELECTRICAL_CABINET".PS_24V_NOT_READY_DEV_ALARM_1 AND NOT "DB2120_MPP_ITC_IPC".RESET_FAULTS);
   "DB426_ALARMS_WARNINGS".ALARMS.GENERAL."702703" := "DB2103_ELECTRICAL_CABINET".PS_24V_NOT_READY_DEV_ALARM_1;
END_REGION

REGION Network 22: POWER SUPPLY 24V NOT READY DEVICE 2 ALARM
   RUNG wire#powerrail
      Contact( "DB2103_ELECTRICAL_CABINET".INPUT_PS_24V_NOT_READY_DEV_2 )
      wire#w1
      Coil( "DB2103_ELECTRICAL_CABINET".PS_24V_NOT_READY_DEV_ALARM_2 )
   END_RUNG
   RUNG wire#powerrail
      Contact( "DB2103_ELECTRICAL_CABINET".PS_24V_NOT_READY_DEV_ALARM_2 )
      I_Contact( "DB2120_MPP_ITC_IPC".RESET_FAULTS )
   END_RUNG wire#w1
   RUNG wire#w1
      Coil( "DB426_ALARMS_WARNINGS".ALARMS.GENERAL."702704" )
   END_RUNG
   // the same network as SCL:
   "DB2103_ELECTRICAL_CABINET".PS_24V_NOT_READY_DEV_ALARM_2 := "DB2103_ELECTRICAL_CABINET".INPUT_PS_24V_NOT_READY_DEV_2 OR ("DB2103_ELECTRICAL_CABINET".PS_24V_NOT_READY_DEV_ALARM_2 AND NOT "DB2120_MPP_ITC_IPC".RESET_FAULTS);
   "DB426_ALARMS_WARNINGS".ALARMS.GENERAL."702704" := "DB2103_ELECTRICAL_CABINET".PS_24V_NOT_READY_DEV_ALARM_2;
END_REGION

REGION Network 23: POWER SUPPLY 24V NOT READY DEVICE 3 ALARM
   RUNG wire#powerrail
      Contact( "DB2103_ELECTRICAL_CABINET".INPUT_PS_24V_NOT_READY_DEV_3 )
      wire#w1
      Coil( "DB2103_ELECTRICAL_CABINET".PS_24V_NOT_READY_DEV_ALARM_3 )
   END_RUNG
   RUNG wire#powerrail
      Contact( "DB2103_ELECTRICAL_CABINET".PS_24V_NOT_READY_DEV_ALARM_3 )
      I_Contact( "DB2120_MPP_ITC_IPC".RESET_FAULTS )
   END_RUNG wire#w1
   RUNG wire#w1
      Coil( "DB426_ALARMS_WARNINGS".ALARMS.GENERAL."702705" )
   END_RUNG
   // the same network as SCL:
   "DB2103_ELECTRICAL_CABINET".PS_24V_NOT_READY_DEV_ALARM_3 := "DB2103_ELECTRICAL_CABINET".INPUT_PS_24V_NOT_READY_DEV_3 OR ("DB2103_ELECTRICAL_CABINET".PS_24V_NOT_READY_DEV_ALARM_3 AND NOT "DB2120_MPP_ITC_IPC".RESET_FAULTS);
   "DB426_ALARMS_WARNINGS".ALARMS.GENERAL."702705" := "DB2103_ELECTRICAL_CABINET".PS_24V_NOT_READY_DEV_ALARM_3;
END_REGION

REGION Network 24: POWER SUPPLY 24V NOT READY DEVICE 4 ALARM
   RUNG wire#powerrail
      Contact( "DB2103_ELECTRICAL_CABINET".INPUT_PS_24V_NOT_READY_DEV_4 )
      wire#w1
      Coil( "DB2103_ELECTRICAL_CABINET".PS_24V_NOT_READY_DEV_ALARM_4 )
   END_RUNG
   RUNG wire#powerrail
      Contact( "DB2103_ELECTRICAL_CABINET".PS_24V_NOT_READY_DEV_ALARM_4 )
      I_Contact( "DB2120_MPP_ITC_IPC".RESET_FAULTS )
   END_RUNG wire#w1
   RUNG wire#w1
      Coil( "DB426_ALARMS_WARNINGS".ALARMS.GENERAL."702706" )
   END_RUNG
   // the same network as SCL:
   "DB2103_ELECTRICAL_CABINET".PS_24V_NOT_READY_DEV_ALARM_4 := "DB2103_ELECTRICAL_CABINET".INPUT_PS_24V_NOT_READY_DEV_4 OR ("DB2103_ELECTRICAL_CABINET".PS_24V_NOT_READY_DEV_ALARM_4 AND NOT "DB2120_MPP_ITC_IPC".RESET_FAULTS);
   "DB426_ALARMS_WARNINGS".ALARMS.GENERAL."702706" := "DB2103_ELECTRICAL_CABINET".PS_24V_NOT_READY_DEV_ALARM_4;
END_REGION

REGION Network 25: POWER SUPPLY 24V NOT READY DEVICE 5 ALARM
   RUNG wire#powerrail
      Contact( "DB2103_ELECTRICAL_CABINET".INPUT_PS_24V_NOT_READY_DEV_5 )
      wire#w1
      Coil( "DB2103_ELECTRICAL_CABINET".PS_24V_NOT_READY_DEV_ALARM_5 )
   END_RUNG
   RUNG wire#powerrail
      Contact( "DB2103_ELECTRICAL_CABINET".PS_24V_NOT_READY_DEV_ALARM_5 )
      I_Contact( "DB2120_MPP_ITC_IPC".RESET_FAULTS )
   END_RUNG wire#w1
   RUNG wire#w1
      Coil( "DB426_ALARMS_WARNINGS".ALARMS.GENERAL."702707" )
   END_RUNG
   // the same network as SCL:
   "DB2103_ELECTRICAL_CABINET".PS_24V_NOT_READY_DEV_ALARM_5 := "DB2103_ELECTRICAL_CABINET".INPUT_PS_24V_NOT_READY_DEV_5 OR ("DB2103_ELECTRICAL_CABINET".PS_24V_NOT_READY_DEV_ALARM_5 AND NOT "DB2120_MPP_ITC_IPC".RESET_FAULTS);
   "DB426_ALARMS_WARNINGS".ALARMS.GENERAL."702707" := "DB2103_ELECTRICAL_CABINET".PS_24V_NOT_READY_DEV_ALARM_5;
END_REGION

REGION Network 26: POWER SUPPLY 24V NOT READY DEVICE 6 ALARM
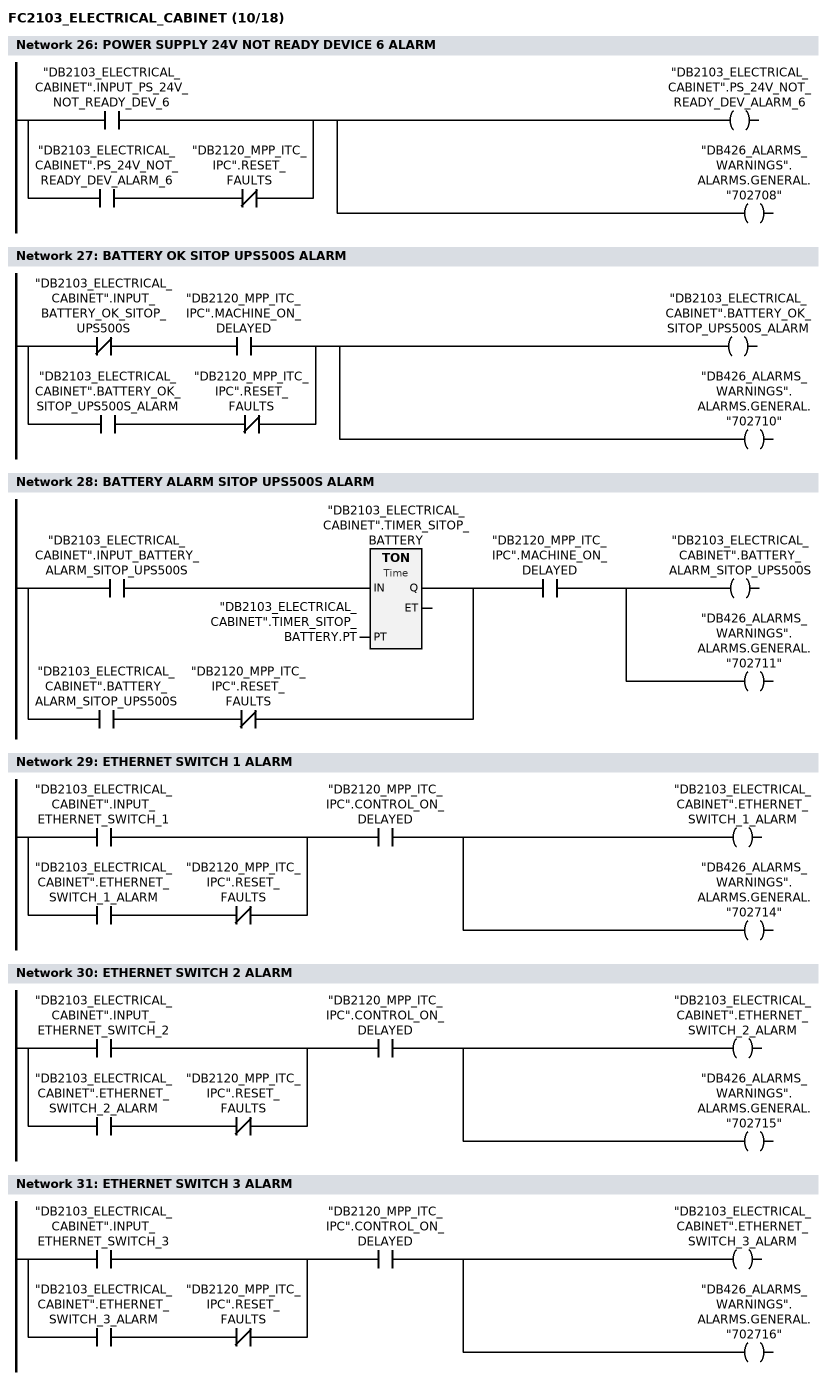
   RUNG wire#powerrail
      Contact( "DB2103_ELECTRICAL_CABINET".INPUT_PS_24V_NOT_READY_DEV_6 )
      wire#w1
      Coil( "DB2103_ELECTRICAL_CABINET".PS_24V_NOT_READY_DEV_ALARM_6 )
   END_RUNG
   RUNG wire#powerrail
      Contact( "DB2103_ELECTRICAL_CABINET".PS_24V_NOT_READY_DEV_ALARM_6 )
      I_Contact( "DB2120_MPP_ITC_IPC".RESET_FAULTS )
   END_RUNG wire#w1
   RUNG wire#w1
      Coil( "DB426_ALARMS_WARNINGS".ALARMS.GENERAL."702708" )
   END_RUNG
   // the same network as SCL:
   "DB2103_ELECTRICAL_CABINET".PS_24V_NOT_READY_DEV_ALARM_6 := "DB2103_ELECTRICAL_CABINET".INPUT_PS_24V_NOT_READY_DEV_6 OR ("DB2103_ELECTRICAL_CABINET".PS_24V_NOT_READY_DEV_ALARM_6 AND NOT "DB2120_MPP_ITC_IPC".RESET_FAULTS);
   "DB426_ALARMS_WARNINGS".ALARMS.GENERAL."702708" := "DB2103_ELECTRICAL_CABINET".PS_24V_NOT_READY_DEV_ALARM_6;
END_REGION

REGION Network 27: BATTERY OK SITOP UPS500S ALARM
   RUNG wire#powerrail
      I_Contact( "DB2103_ELECTRICAL_CABINET".INPUT_BATTERY_OK_SITOP_UPS500S )
      Contact( "DB2120_MPP_ITC_IPC".MACHINE_ON_DELAYED )
      wire#w1
      Coil( "DB2103_ELECTRICAL_CABINET".BATTERY_OK_SITOP_UPS500S_ALARM )
   END_RUNG
   RUNG wire#powerrail
      Contact( "DB2103_ELECTRICAL_CABINET".BATTERY_OK_SITOP_UPS500S_ALARM )
      I_Contact( "DB2120_MPP_ITC_IPC".RESET_FAULTS )
   END_RUNG wire#w1
   RUNG wire#w1
      Coil( "DB426_ALARMS_WARNINGS".ALARMS.GENERAL."702710" )
   END_RUNG
   // the same network as SCL:
   "DB2103_ELECTRICAL_CABINET".BATTERY_OK_SITOP_UPS500S_ALARM := (NOT "DB2103_ELECTRICAL_CABINET".INPUT_BATTERY_OK_SITOP_UPS500S AND "DB2120_MPP_ITC_IPC".MACHINE_ON_DELAYED) OR ("DB2103_ELECTRICAL_CABINET".BATTERY_OK_SITOP_UPS500S_ALARM AND NOT "DB2120_MPP_ITC_IPC".RESET_FAULTS);
   "DB426_ALARMS_WARNINGS".ALARMS.GENERAL."702710" := "DB2103_ELECTRICAL_CABINET".BATTERY_OK_SITOP_UPS500S_ALARM;
END_REGION

REGION Network 28: BATTERY ALARM SITOP UPS500S ALARM
   RUNG wire#powerrail
      Contact( "DB2103_ELECTRICAL_CABINET".INPUT_BATTERY_ALARM_SITOP_UPS500S )
      { S7_Templates := "time_type := Time" } "DB2103_ELECTRICAL_CABINET".TIMER_SITOP_BATTERY.TON(pt := "DB2103_ELECTRICAL_CABINET".TIMER_SITOP_BATTERY.PT, et =>)
      wire#w1
      Contact( "DB2120_MPP_ITC_IPC".MACHINE_ON_DELAYED )
      wire#w2
      Coil( "DB2103_ELECTRICAL_CABINET".BATTERY_ALARM_SITOP_UPS500S )
   END_RUNG
   RUNG wire#powerrail
      Contact( "DB2103_ELECTRICAL_CABINET".BATTERY_ALARM_SITOP_UPS500S )
      I_Contact( "DB2120_MPP_ITC_IPC".RESET_FAULTS )
   END_RUNG wire#w1
   RUNG wire#w2
      Coil( "DB426_ALARMS_WARNINGS".ALARMS.GENERAL."702711" )
   END_RUNG
   // the same network as SCL:
   "DB2103_ELECTRICAL_CABINET".TIMER_SITOP_BATTERY.TON(IN := "DB2103_ELECTRICAL_CABINET".INPUT_BATTERY_ALARM_SITOP_UPS500S,
                           PT := "DB2103_ELECTRICAL_CABINET".TIMER_SITOP_BATTERY.PT);
   "DB2103_ELECTRICAL_CABINET".BATTERY_ALARM_SITOP_UPS500S := ("DB2103_ELECTRICAL_CABINET".TIMER_SITOP_BATTERY.Q OR ("DB2103_ELECTRICAL_CABINET".BATTERY_ALARM_SITOP_UPS500S AND NOT "DB2120_MPP_ITC_IPC".RESET_FAULTS)) AND "DB2120_MPP_ITC_IPC".MACHINE_ON_DELAYED;
   "DB426_ALARMS_WARNINGS".ALARMS.GENERAL."702711" := "DB2103_ELECTRICAL_CABINET".BATTERY_ALARM_SITOP_UPS500S;
END_REGION

REGION Network 29: ETHERNET SWITCH 1 ALARM
   RUNG wire#powerrail
      Contact( "DB2103_ELECTRICAL_CABINET".INPUT_ETHERNET_SWITCH_1 )
      wire#w1
      Contact( "DB2120_MPP_ITC_IPC".CONTROL_ON_DELAYED )
      wire#w2
      Coil( "DB2103_ELECTRICAL_CABINET".ETHERNET_SWITCH_1_ALARM )
   END_RUNG
   RUNG wire#powerrail
      Contact( "DB2103_ELECTRICAL_CABINET".ETHERNET_SWITCH_1_ALARM )
      I_Contact( "DB2120_MPP_ITC_IPC".RESET_FAULTS )
   END_RUNG wire#w1
   RUNG wire#w2
      Coil( "DB426_ALARMS_WARNINGS".ALARMS.GENERAL."702714" )
   END_RUNG
   // the same network as SCL:
   "DB2103_ELECTRICAL_CABINET".ETHERNET_SWITCH_1_ALARM := ("DB2103_ELECTRICAL_CABINET".INPUT_ETHERNET_SWITCH_1 OR ("DB2103_ELECTRICAL_CABINET".ETHERNET_SWITCH_1_ALARM AND NOT "DB2120_MPP_ITC_IPC".RESET_FAULTS)) AND "DB2120_MPP_ITC_IPC".CONTROL_ON_DELAYED;
   "DB426_ALARMS_WARNINGS".ALARMS.GENERAL."702714" := "DB2103_ELECTRICAL_CABINET".ETHERNET_SWITCH_1_ALARM;
END_REGION

REGION Network 30: ETHERNET SWITCH 2 ALARM
   RUNG wire#powerrail
      Contact( "DB2103_ELECTRICAL_CABINET".INPUT_ETHERNET_SWITCH_2 )
      wire#w1
      Contact( "DB2120_MPP_ITC_IPC".CONTROL_ON_DELAYED )
      wire#w2
      Coil( "DB2103_ELECTRICAL_CABINET".ETHERNET_SWITCH_2_ALARM )
   END_RUNG
   RUNG wire#powerrail
      Contact( "DB2103_ELECTRICAL_CABINET".ETHERNET_SWITCH_2_ALARM )
      I_Contact( "DB2120_MPP_ITC_IPC".RESET_FAULTS )
   END_RUNG wire#w1
   RUNG wire#w2
      Coil( "DB426_ALARMS_WARNINGS".ALARMS.GENERAL."702715" )
   END_RUNG
   // the same network as SCL:
   "DB2103_ELECTRICAL_CABINET".ETHERNET_SWITCH_2_ALARM := ("DB2103_ELECTRICAL_CABINET".INPUT_ETHERNET_SWITCH_2 OR ("DB2103_ELECTRICAL_CABINET".ETHERNET_SWITCH_2_ALARM AND NOT "DB2120_MPP_ITC_IPC".RESET_FAULTS)) AND "DB2120_MPP_ITC_IPC".CONTROL_ON_DELAYED;
   "DB426_ALARMS_WARNINGS".ALARMS.GENERAL."702715" := "DB2103_ELECTRICAL_CABINET".ETHERNET_SWITCH_2_ALARM;
END_REGION

REGION Network 31: ETHERNET SWITCH 3 ALARM
   RUNG wire#powerrail
      Contact( "DB2103_ELECTRICAL_CABINET".INPUT_ETHERNET_SWITCH_3 )
      wire#w1
      Contact( "DB2120_MPP_ITC_IPC".CONTROL_ON_DELAYED )
      wire#w2
      Coil( "DB2103_ELECTRICAL_CABINET".ETHERNET_SWITCH_3_ALARM )
   END_RUNG
   RUNG wire#powerrail
      Contact( "DB2103_ELECTRICAL_CABINET".ETHERNET_SWITCH_3_ALARM )
      I_Contact( "DB2120_MPP_ITC_IPC".RESET_FAULTS )
   END_RUNG wire#w1
   RUNG wire#w2
      Coil( "DB426_ALARMS_WARNINGS".ALARMS.GENERAL."702716" )
   END_RUNG
   // the same network as SCL:
   "DB2103_ELECTRICAL_CABINET".ETHERNET_SWITCH_3_ALARM := ("DB2103_ELECTRICAL_CABINET".INPUT_ETHERNET_SWITCH_3 OR ("DB2103_ELECTRICAL_CABINET".ETHERNET_SWITCH_3_ALARM AND NOT "DB2120_MPP_ITC_IPC".RESET_FAULTS)) AND "DB2120_MPP_ITC_IPC".CONTROL_ON_DELAYED;
   "DB426_ALARMS_WARNINGS".ALARMS.GENERAL."702716" := "DB2103_ELECTRICAL_CABINET".ETHERNET_SWITCH_3_ALARM;
END_REGION

REGION Network 32: PROFINET CONTROL UNIT FAULT ALARM
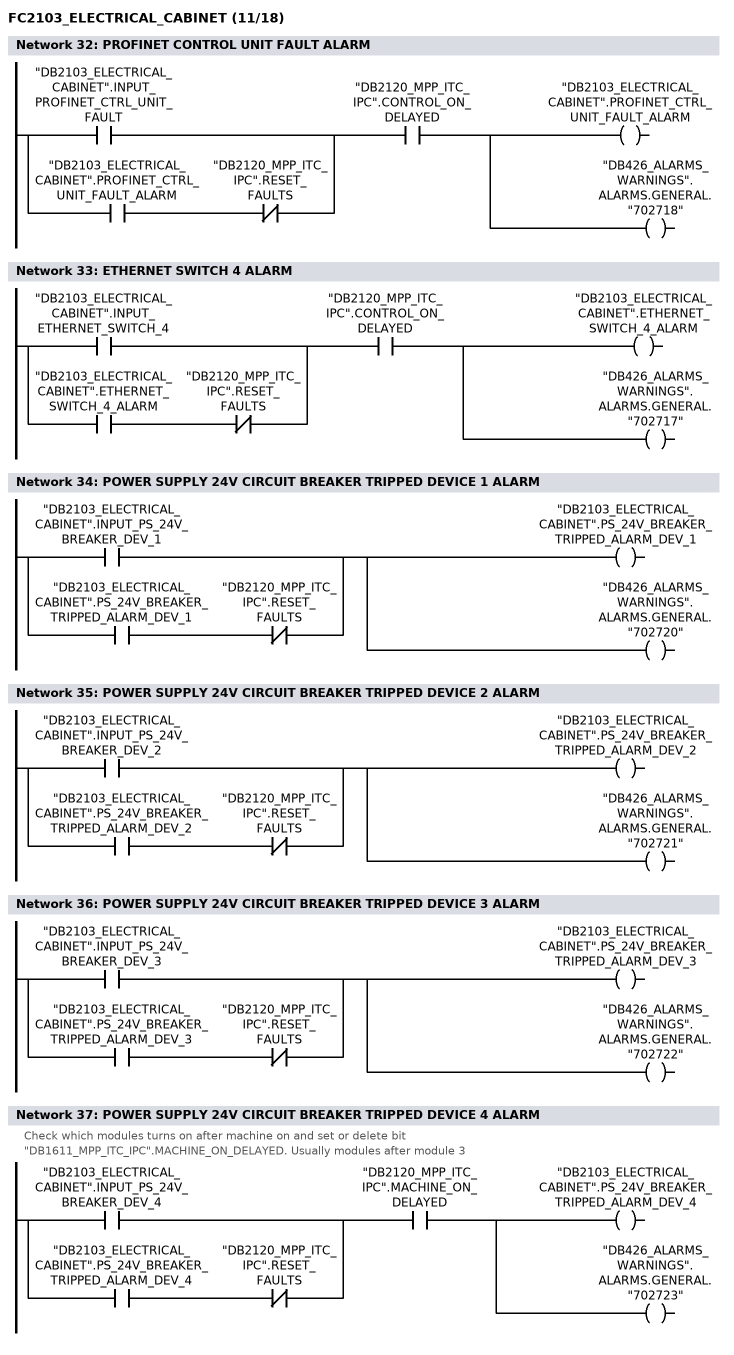
   RUNG wire#powerrail
      Contact( "DB2103_ELECTRICAL_CABINET".INPUT_PROFINET_CTRL_UNIT_FAULT )
      wire#w1
      Contact( "DB2120_MPP_ITC_IPC".CONTROL_ON_DELAYED )
      wire#w2
      Coil( "DB2103_ELECTRICAL_CABINET".PROFINET_CTRL_UNIT_FAULT_ALARM )
   END_RUNG
   RUNG wire#powerrail
      Contact( "DB2103_ELECTRICAL_CABINET".PROFINET_CTRL_UNIT_FAULT_ALARM )
      I_Contact( "DB2120_MPP_ITC_IPC".RESET_FAULTS )
   END_RUNG wire#w1
   RUNG wire#w2
      Coil( "DB426_ALARMS_WARNINGS".ALARMS.GENERAL."702718" )
   END_RUNG
   // the same network as SCL:
   "DB2103_ELECTRICAL_CABINET".PROFINET_CTRL_UNIT_FAULT_ALARM := ("DB2103_ELECTRICAL_CABINET".INPUT_PROFINET_CTRL_UNIT_FAULT OR ("DB2103_ELECTRICAL_CABINET".PROFINET_CTRL_UNIT_FAULT_ALARM AND NOT "DB2120_MPP_ITC_IPC".RESET_FAULTS)) AND "DB2120_MPP_ITC_IPC".CONTROL_ON_DELAYED;
   "DB426_ALARMS_WARNINGS".ALARMS.GENERAL."702718" := "DB2103_ELECTRICAL_CABINET".PROFINET_CTRL_UNIT_FAULT_ALARM;
END_REGION

REGION Network 33: ETHERNET SWITCH 4 ALARM
   RUNG wire#powerrail
      Contact( "DB2103_ELECTRICAL_CABINET".INPUT_ETHERNET_SWITCH_4 )
      wire#w1
      Contact( "DB2120_MPP_ITC_IPC".CONTROL_ON_DELAYED )
      wire#w2
      Coil( "DB2103_ELECTRICAL_CABINET".ETHERNET_SWITCH_4_ALARM )
   END_RUNG
   RUNG wire#powerrail
      Contact( "DB2103_ELECTRICAL_CABINET".ETHERNET_SWITCH_4_ALARM )
      I_Contact( "DB2120_MPP_ITC_IPC".RESET_FAULTS )
   END_RUNG wire#w1
   RUNG wire#w2
      Coil( "DB426_ALARMS_WARNINGS".ALARMS.GENERAL."702717" )
   END_RUNG
   // the same network as SCL:
   "DB2103_ELECTRICAL_CABINET".ETHERNET_SWITCH_4_ALARM := ("DB2103_ELECTRICAL_CABINET".INPUT_ETHERNET_SWITCH_4 OR ("DB2103_ELECTRICAL_CABINET".ETHERNET_SWITCH_4_ALARM AND NOT "DB2120_MPP_ITC_IPC".RESET_FAULTS)) AND "DB2120_MPP_ITC_IPC".CONTROL_ON_DELAYED;
   "DB426_ALARMS_WARNINGS".ALARMS.GENERAL."702717" := "DB2103_ELECTRICAL_CABINET".ETHERNET_SWITCH_4_ALARM;
END_REGION

REGION Network 34: POWER SUPPLY 24V CIRCUIT BREAKER TRIPPED DEVICE 1 ALARM
   RUNG wire#powerrail
      Contact( "DB2103_ELECTRICAL_CABINET".INPUT_PS_24V_BREAKER_DEV_1 )
      wire#w1
      Coil( "DB2103_ELECTRICAL_CABINET".PS_24V_BREAKER_TRIPPED_ALARM_DEV_1 )
   END_RUNG
   RUNG wire#powerrail
      Contact( "DB2103_ELECTRICAL_CABINET".PS_24V_BREAKER_TRIPPED_ALARM_DEV_1 )
      I_Contact( "DB2120_MPP_ITC_IPC".RESET_FAULTS )
   END_RUNG wire#w1
   RUNG wire#w1
      Coil( "DB426_ALARMS_WARNINGS".ALARMS.GENERAL."702720" )
   END_RUNG
   // the same network as SCL:
   "DB2103_ELECTRICAL_CABINET".PS_24V_BREAKER_TRIPPED_ALARM_DEV_1 := "DB2103_ELECTRICAL_CABINET".INPUT_PS_24V_BREAKER_DEV_1 OR ("DB2103_ELECTRICAL_CABINET".PS_24V_BREAKER_TRIPPED_ALARM_DEV_1 AND NOT "DB2120_MPP_ITC_IPC".RESET_FAULTS);
   "DB426_ALARMS_WARNINGS".ALARMS.GENERAL."702720" := "DB2103_ELECTRICAL_CABINET".PS_24V_BREAKER_TRIPPED_ALARM_DEV_1;
END_REGION

REGION Network 35: POWER SUPPLY 24V CIRCUIT BREAKER TRIPPED DEVICE 2 ALARM
   RUNG wire#powerrail
      Contact( "DB2103_ELECTRICAL_CABINET".INPUT_PS_24V_BREAKER_DEV_2 )
      wire#w1
      Coil( "DB2103_ELECTRICAL_CABINET".PS_24V_BREAKER_TRIPPED_ALARM_DEV_2 )
   END_RUNG
   RUNG wire#powerrail
      Contact( "DB2103_ELECTRICAL_CABINET".PS_24V_BREAKER_TRIPPED_ALARM_DEV_2 )
      I_Contact( "DB2120_MPP_ITC_IPC".RESET_FAULTS )
   END_RUNG wire#w1
   RUNG wire#w1
      Coil( "DB426_ALARMS_WARNINGS".ALARMS.GENERAL."702721" )
   END_RUNG
   // the same network as SCL:
   "DB2103_ELECTRICAL_CABINET".PS_24V_BREAKER_TRIPPED_ALARM_DEV_2 := "DB2103_ELECTRICAL_CABINET".INPUT_PS_24V_BREAKER_DEV_2 OR ("DB2103_ELECTRICAL_CABINET".PS_24V_BREAKER_TRIPPED_ALARM_DEV_2 AND NOT "DB2120_MPP_ITC_IPC".RESET_FAULTS);
   "DB426_ALARMS_WARNINGS".ALARMS.GENERAL."702721" := "DB2103_ELECTRICAL_CABINET".PS_24V_BREAKER_TRIPPED_ALARM_DEV_2;
END_REGION

REGION Network 36: POWER SUPPLY 24V CIRCUIT BREAKER TRIPPED DEVICE 3 ALARM
   RUNG wire#powerrail
      Contact( "DB2103_ELECTRICAL_CABINET".INPUT_PS_24V_BREAKER_DEV_3 )
      wire#w1
      Coil( "DB2103_ELECTRICAL_CABINET".PS_24V_BREAKER_TRIPPED_ALARM_DEV_3 )
   END_RUNG
   RUNG wire#powerrail
      Contact( "DB2103_ELECTRICAL_CABINET".PS_24V_BREAKER_TRIPPED_ALARM_DEV_3 )
      I_Contact( "DB2120_MPP_ITC_IPC".RESET_FAULTS )
   END_RUNG wire#w1
   RUNG wire#w1
      Coil( "DB426_ALARMS_WARNINGS".ALARMS.GENERAL."702722" )
   END_RUNG
   // the same network as SCL:
   "DB2103_ELECTRICAL_CABINET".PS_24V_BREAKER_TRIPPED_ALARM_DEV_3 := "DB2103_ELECTRICAL_CABINET".INPUT_PS_24V_BREAKER_DEV_3 OR ("DB2103_ELECTRICAL_CABINET".PS_24V_BREAKER_TRIPPED_ALARM_DEV_3 AND NOT "DB2120_MPP_ITC_IPC".RESET_FAULTS);
   "DB426_ALARMS_WARNINGS".ALARMS.GENERAL."702722" := "DB2103_ELECTRICAL_CABINET".PS_24V_BREAKER_TRIPPED_ALARM_DEV_3;
END_REGION

REGION Network 37: POWER SUPPLY 24V CIRCUIT BREAKER TRIPPED DEVICE 4 ALARM
   // Check which modules turns on after machine on and set or delete bit 
   // "DB1611_MPP_ITC_IPC".MACHINE_ON_DELAYED. Usually modules after module 3
   RUNG wire#powerrail
      Contact( "DB2103_ELECTRICAL_CABINET".INPUT_PS_24V_BREAKER_DEV_4 )
      wire#w1
      Contact( "DB2120_MPP_ITC_IPC".MACHINE_ON_DELAYED )
      wire#w2
      Coil( "DB2103_ELECTRICAL_CABINET".PS_24V_BREAKER_TRIPPED_ALARM_DEV_4 )
   END_RUNG
   RUNG wire#powerrail
      Contact( "DB2103_ELECTRICAL_CABINET".PS_24V_BREAKER_TRIPPED_ALARM_DEV_4 )
      I_Contact( "DB2120_MPP_ITC_IPC".RESET_FAULTS )
   END_RUNG wire#w1
   RUNG wire#w2
      Coil( "DB426_ALARMS_WARNINGS".ALARMS.GENERAL."702723" )
   END_RUNG
   // the same network as SCL:
   "DB2103_ELECTRICAL_CABINET".PS_24V_BREAKER_TRIPPED_ALARM_DEV_4 := ("DB2103_ELECTRICAL_CABINET".INPUT_PS_24V_BREAKER_DEV_4 OR ("DB2103_ELECTRICAL_CABINET".PS_24V_BREAKER_TRIPPED_ALARM_DEV_4 AND NOT "DB2120_MPP_ITC_IPC".RESET_FAULTS)) AND "DB2120_MPP_ITC_IPC".MACHINE_ON_DELAYED;
   "DB426_ALARMS_WARNINGS".ALARMS.GENERAL."702723" := "DB2103_ELECTRICAL_CABINET".PS_24V_BREAKER_TRIPPED_ALARM_DEV_4;
END_REGION

REGION Network 38: SINAMICS CIRCUIT BREAKER TRIPPED ALARM
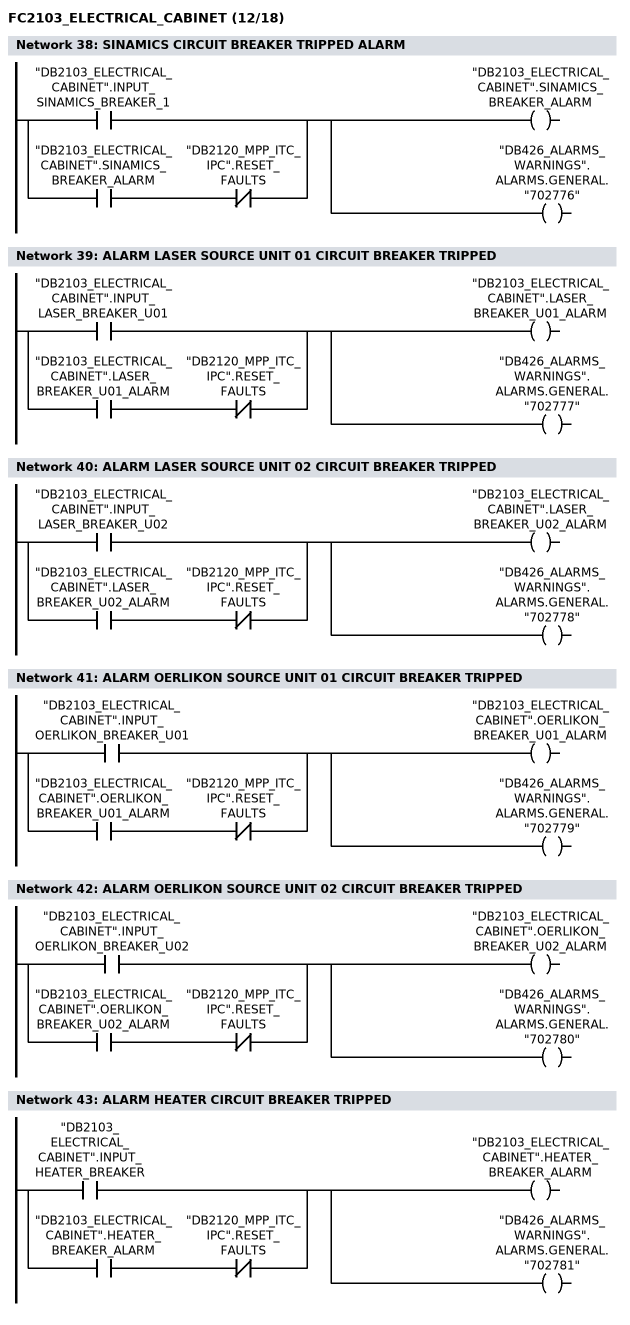
   RUNG wire#powerrail
      Contact( "DB2103_ELECTRICAL_CABINET".INPUT_SINAMICS_BREAKER_1 )
      wire#w1
      Coil( "DB2103_ELECTRICAL_CABINET".SINAMICS_BREAKER_ALARM )
   END_RUNG
   RUNG wire#powerrail
      Contact( "DB2103_ELECTRICAL_CABINET".SINAMICS_BREAKER_ALARM )
      I_Contact( "DB2120_MPP_ITC_IPC".RESET_FAULTS )
   END_RUNG wire#w1
   RUNG wire#w1
      Coil( "DB426_ALARMS_WARNINGS".ALARMS.GENERAL."702776" )
   END_RUNG
   // the same network as SCL:
   "DB2103_ELECTRICAL_CABINET".SINAMICS_BREAKER_ALARM := "DB2103_ELECTRICAL_CABINET".INPUT_SINAMICS_BREAKER_1 OR ("DB2103_ELECTRICAL_CABINET".SINAMICS_BREAKER_ALARM AND NOT "DB2120_MPP_ITC_IPC".RESET_FAULTS);
   "DB426_ALARMS_WARNINGS".ALARMS.GENERAL."702776" := "DB2103_ELECTRICAL_CABINET".SINAMICS_BREAKER_ALARM;
END_REGION

REGION Network 39: ALARM LASER SOURCE UNIT 01 CIRCUIT BREAKER TRIPPED
   RUNG wire#powerrail
      Contact( "DB2103_ELECTRICAL_CABINET".INPUT_LASER_BREAKER_U01 )
      wire#w1
      Coil( "DB2103_ELECTRICAL_CABINET".LASER_BREAKER_U01_ALARM )
   END_RUNG
   RUNG wire#powerrail
      Contact( "DB2103_ELECTRICAL_CABINET".LASER_BREAKER_U01_ALARM )
      I_Contact( "DB2120_MPP_ITC_IPC".RESET_FAULTS )
   END_RUNG wire#w1
   RUNG wire#w1
      Coil( "DB426_ALARMS_WARNINGS".ALARMS.GENERAL."702777" )
   END_RUNG
   // the same network as SCL:
   "DB2103_ELECTRICAL_CABINET".LASER_BREAKER_U01_ALARM := "DB2103_ELECTRICAL_CABINET".INPUT_LASER_BREAKER_U01 OR ("DB2103_ELECTRICAL_CABINET".LASER_BREAKER_U01_ALARM AND NOT "DB2120_MPP_ITC_IPC".RESET_FAULTS);
   "DB426_ALARMS_WARNINGS".ALARMS.GENERAL."702777" := "DB2103_ELECTRICAL_CABINET".LASER_BREAKER_U01_ALARM;
END_REGION

REGION Network 40: ALARM LASER SOURCE UNIT 02 CIRCUIT BREAKER TRIPPED
   RUNG wire#powerrail
      Contact( "DB2103_ELECTRICAL_CABINET".INPUT_LASER_BREAKER_U02 )
      wire#w1
      Coil( "DB2103_ELECTRICAL_CABINET".LASER_BREAKER_U02_ALARM )
   END_RUNG
   RUNG wire#powerrail
      Contact( "DB2103_ELECTRICAL_CABINET".LASER_BREAKER_U02_ALARM )
      I_Contact( "DB2120_MPP_ITC_IPC".RESET_FAULTS )
   END_RUNG wire#w1
   RUNG wire#w1
      Coil( "DB426_ALARMS_WARNINGS".ALARMS.GENERAL."702778" )
   END_RUNG
   // the same network as SCL:
   "DB2103_ELECTRICAL_CABINET".LASER_BREAKER_U02_ALARM := "DB2103_ELECTRICAL_CABINET".INPUT_LASER_BREAKER_U02 OR ("DB2103_ELECTRICAL_CABINET".LASER_BREAKER_U02_ALARM AND NOT "DB2120_MPP_ITC_IPC".RESET_FAULTS);
   "DB426_ALARMS_WARNINGS".ALARMS.GENERAL."702778" := "DB2103_ELECTRICAL_CABINET".LASER_BREAKER_U02_ALARM;
END_REGION

REGION Network 41: ALARM OERLIKON SOURCE UNIT 01 CIRCUIT BREAKER TRIPPED
   RUNG wire#powerrail
      Contact( "DB2103_ELECTRICAL_CABINET".INPUT_OERLIKON_BREAKER_U01 )
      wire#w1
      Coil( "DB2103_ELECTRICAL_CABINET".OERLIKON_BREAKER_U01_ALARM )
   END_RUNG
   RUNG wire#powerrail
      Contact( "DB2103_ELECTRICAL_CABINET".OERLIKON_BREAKER_U01_ALARM )
      I_Contact( "DB2120_MPP_ITC_IPC".RESET_FAULTS )
   END_RUNG wire#w1
   RUNG wire#w1
      Coil( "DB426_ALARMS_WARNINGS".ALARMS.GENERAL."702779" )
   END_RUNG
   // the same network as SCL:
   "DB2103_ELECTRICAL_CABINET".OERLIKON_BREAKER_U01_ALARM := "DB2103_ELECTRICAL_CABINET".INPUT_OERLIKON_BREAKER_U01 OR ("DB2103_ELECTRICAL_CABINET".OERLIKON_BREAKER_U01_ALARM AND NOT "DB2120_MPP_ITC_IPC".RESET_FAULTS);
   "DB426_ALARMS_WARNINGS".ALARMS.GENERAL."702779" := "DB2103_ELECTRICAL_CABINET".OERLIKON_BREAKER_U01_ALARM;
END_REGION

REGION Network 42: ALARM OERLIKON SOURCE UNIT 02 CIRCUIT BREAKER TRIPPED
   RUNG wire#powerrail
      Contact( "DB2103_ELECTRICAL_CABINET".INPUT_OERLIKON_BREAKER_U02 )
      wire#w1
      Coil( "DB2103_ELECTRICAL_CABINET".OERLIKON_BREAKER_U02_ALARM )
   END_RUNG
   RUNG wire#powerrail
      Contact( "DB2103_ELECTRICAL_CABINET".OERLIKON_BREAKER_U02_ALARM )
      I_Contact( "DB2120_MPP_ITC_IPC".RESET_FAULTS )
   END_RUNG wire#w1
   RUNG wire#w1
      Coil( "DB426_ALARMS_WARNINGS".ALARMS.GENERAL."702780" )
   END_RUNG
   // the same network as SCL:
   "DB2103_ELECTRICAL_CABINET".OERLIKON_BREAKER_U02_ALARM := "DB2103_ELECTRICAL_CABINET".INPUT_OERLIKON_BREAKER_U02 OR ("DB2103_ELECTRICAL_CABINET".OERLIKON_BREAKER_U02_ALARM AND NOT "DB2120_MPP_ITC_IPC".RESET_FAULTS);
   "DB426_ALARMS_WARNINGS".ALARMS.GENERAL."702780" := "DB2103_ELECTRICAL_CABINET".OERLIKON_BREAKER_U02_ALARM;
END_REGION

REGION Network 43: ALARM HEATER CIRCUIT BREAKER TRIPPED
   RUNG wire#powerrail
      Contact( "DB2103_ELECTRICAL_CABINET".INPUT_HEATER_BREAKER )
      wire#w1
      Coil( "DB2103_ELECTRICAL_CABINET".HEATER_BREAKER_ALARM )
   END_RUNG
   RUNG wire#powerrail
      Contact( "DB2103_ELECTRICAL_CABINET".HEATER_BREAKER_ALARM )
      I_Contact( "DB2120_MPP_ITC_IPC".RESET_FAULTS )
   END_RUNG wire#w1
   RUNG wire#w1
      Coil( "DB426_ALARMS_WARNINGS".ALARMS.GENERAL."702781" )
   END_RUNG
   // the same network as SCL:
   "DB2103_ELECTRICAL_CABINET".HEATER_BREAKER_ALARM := "DB2103_ELECTRICAL_CABINET".INPUT_HEATER_BREAKER OR ("DB2103_ELECTRICAL_CABINET".HEATER_BREAKER_ALARM AND NOT "DB2120_MPP_ITC_IPC".RESET_FAULTS);
   "DB426_ALARMS_WARNINGS".ALARMS.GENERAL."702781" := "DB2103_ELECTRICAL_CABINET".HEATER_BREAKER_ALARM;
END_REGION

REGION Network 44: ALARM STIRRER CIRCUIT BREAKER TRIPPED
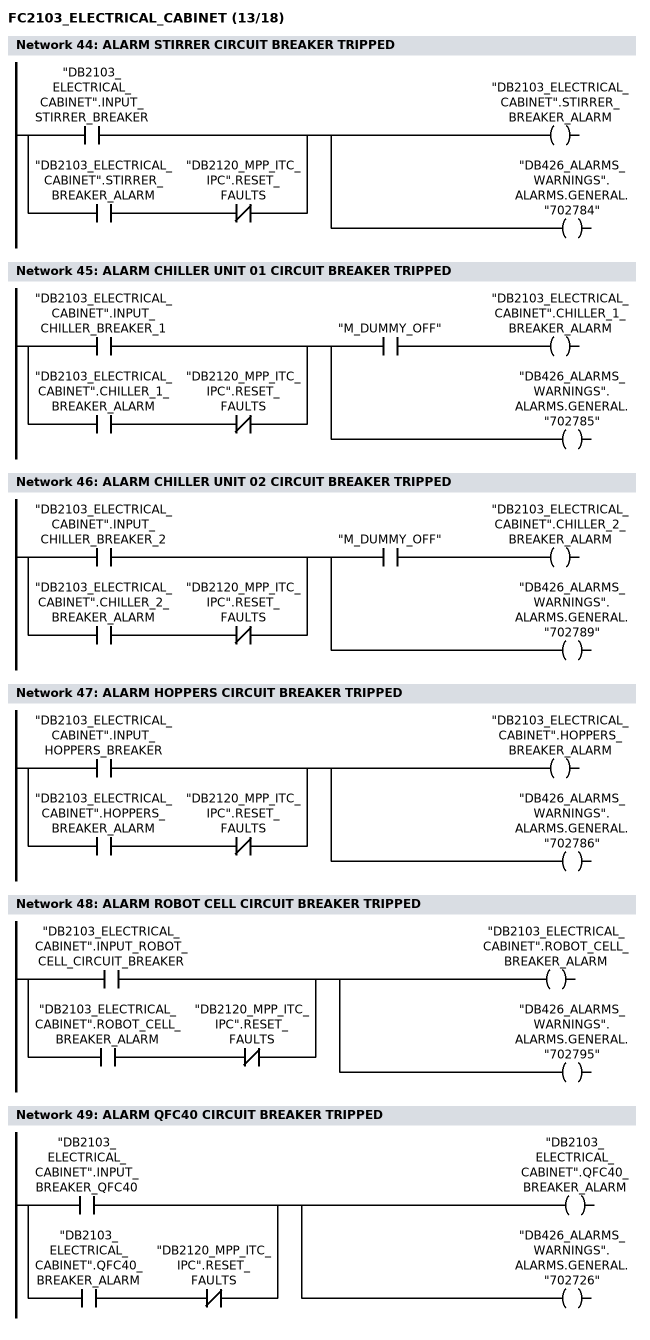
   RUNG wire#powerrail
      Contact( "DB2103_ELECTRICAL_CABINET".INPUT_STIRRER_BREAKER )
      wire#w1
      Coil( "DB2103_ELECTRICAL_CABINET".STIRRER_BREAKER_ALARM )
   END_RUNG
   RUNG wire#powerrail
      Contact( "DB2103_ELECTRICAL_CABINET".STIRRER_BREAKER_ALARM )
      I_Contact( "DB2120_MPP_ITC_IPC".RESET_FAULTS )
   END_RUNG wire#w1
   RUNG wire#w1
      Coil( "DB426_ALARMS_WARNINGS".ALARMS.GENERAL."702784" )
   END_RUNG
   // the same network as SCL:
   "DB2103_ELECTRICAL_CABINET".STIRRER_BREAKER_ALARM := "DB2103_ELECTRICAL_CABINET".INPUT_STIRRER_BREAKER OR ("DB2103_ELECTRICAL_CABINET".STIRRER_BREAKER_ALARM AND NOT "DB2120_MPP_ITC_IPC".RESET_FAULTS);
   "DB426_ALARMS_WARNINGS".ALARMS.GENERAL."702784" := "DB2103_ELECTRICAL_CABINET".STIRRER_BREAKER_ALARM;
END_REGION

REGION Network 45: ALARM CHILLER UNIT 01 CIRCUIT BREAKER TRIPPED
   RUNG wire#powerrail
      Contact( "DB2103_ELECTRICAL_CABINET".INPUT_CHILLER_BREAKER_1 )
      wire#w1
      Contact( "M_DUMMY_OFF" )
      Coil( "DB2103_ELECTRICAL_CABINET".CHILLER_1_BREAKER_ALARM )
   END_RUNG
   RUNG wire#powerrail
      Contact( "DB2103_ELECTRICAL_CABINET".CHILLER_1_BREAKER_ALARM )
      I_Contact( "DB2120_MPP_ITC_IPC".RESET_FAULTS )
   END_RUNG wire#w1
   RUNG wire#w1
      Coil( "DB426_ALARMS_WARNINGS".ALARMS.GENERAL."702785" )
   END_RUNG
   // the same network as SCL:
   #_w1 := "DB2103_ELECTRICAL_CABINET".INPUT_CHILLER_BREAKER_1 OR ("DB2103_ELECTRICAL_CABINET".CHILLER_1_BREAKER_ALARM AND NOT "DB2120_MPP_ITC_IPC".RESET_FAULTS);
   "DB2103_ELECTRICAL_CABINET".CHILLER_1_BREAKER_ALARM := #_w1 AND "M_DUMMY_OFF";
   "DB426_ALARMS_WARNINGS".ALARMS.GENERAL."702785" := #_w1;
END_REGION

REGION Network 46: ALARM CHILLER UNIT 02 CIRCUIT BREAKER TRIPPED
   RUNG wire#powerrail
      Contact( "DB2103_ELECTRICAL_CABINET".INPUT_CHILLER_BREAKER_2 )
      wire#w1
      Contact( "M_DUMMY_OFF" )
      Coil( "DB2103_ELECTRICAL_CABINET".CHILLER_2_BREAKER_ALARM )
   END_RUNG
   RUNG wire#powerrail
      Contact( "DB2103_ELECTRICAL_CABINET".CHILLER_2_BREAKER_ALARM )
      I_Contact( "DB2120_MPP_ITC_IPC".RESET_FAULTS )
   END_RUNG wire#w1
   RUNG wire#w1
      Coil( "DB426_ALARMS_WARNINGS".ALARMS.GENERAL."702789" )
   END_RUNG
   // the same network as SCL:
   #_w1 := "DB2103_ELECTRICAL_CABINET".INPUT_CHILLER_BREAKER_2 OR ("DB2103_ELECTRICAL_CABINET".CHILLER_2_BREAKER_ALARM AND NOT "DB2120_MPP_ITC_IPC".RESET_FAULTS);
   "DB2103_ELECTRICAL_CABINET".CHILLER_2_BREAKER_ALARM := #_w1 AND "M_DUMMY_OFF";
   "DB426_ALARMS_WARNINGS".ALARMS.GENERAL."702789" := #_w1;
END_REGION

REGION Network 47: ALARM HOPPERS CIRCUIT BREAKER TRIPPED
   RUNG wire#powerrail
      Contact( "DB2103_ELECTRICAL_CABINET".INPUT_HOPPERS_BREAKER )
      wire#w1
      Coil( "DB2103_ELECTRICAL_CABINET".HOPPERS_BREAKER_ALARM )
   END_RUNG
   RUNG wire#powerrail
      Contact( "DB2103_ELECTRICAL_CABINET".HOPPERS_BREAKER_ALARM )
      I_Contact( "DB2120_MPP_ITC_IPC".RESET_FAULTS )
   END_RUNG wire#w1
   RUNG wire#w1
      Coil( "DB426_ALARMS_WARNINGS".ALARMS.GENERAL."702786" )
   END_RUNG
   // the same network as SCL:
   "DB2103_ELECTRICAL_CABINET".HOPPERS_BREAKER_ALARM := "DB2103_ELECTRICAL_CABINET".INPUT_HOPPERS_BREAKER OR ("DB2103_ELECTRICAL_CABINET".HOPPERS_BREAKER_ALARM AND NOT "DB2120_MPP_ITC_IPC".RESET_FAULTS);
   "DB426_ALARMS_WARNINGS".ALARMS.GENERAL."702786" := "DB2103_ELECTRICAL_CABINET".HOPPERS_BREAKER_ALARM;
END_REGION

REGION Network 48: ALARM ROBOT CELL CIRCUIT BREAKER TRIPPED
   RUNG wire#powerrail
      Contact( "DB2103_ELECTRICAL_CABINET".INPUT_ROBOT_CELL_CIRCUIT_BREAKER )
      wire#w1
      Coil( "DB2103_ELECTRICAL_CABINET".ROBOT_CELL_BREAKER_ALARM )
   END_RUNG
   RUNG wire#powerrail
      Contact( "DB2103_ELECTRICAL_CABINET".ROBOT_CELL_BREAKER_ALARM )
      I_Contact( "DB2120_MPP_ITC_IPC".RESET_FAULTS )
   END_RUNG wire#w1
   RUNG wire#w1
      Coil( "DB426_ALARMS_WARNINGS".ALARMS.GENERAL."702795" )
   END_RUNG
   // the same network as SCL:
   "DB2103_ELECTRICAL_CABINET".ROBOT_CELL_BREAKER_ALARM := "DB2103_ELECTRICAL_CABINET".INPUT_ROBOT_CELL_CIRCUIT_BREAKER OR ("DB2103_ELECTRICAL_CABINET".ROBOT_CELL_BREAKER_ALARM AND NOT "DB2120_MPP_ITC_IPC".RESET_FAULTS);
   "DB426_ALARMS_WARNINGS".ALARMS.GENERAL."702795" := "DB2103_ELECTRICAL_CABINET".ROBOT_CELL_BREAKER_ALARM;
END_REGION

REGION Network 49: ALARM QFC40 CIRCUIT BREAKER TRIPPED
   RUNG wire#powerrail
      Contact( "DB2103_ELECTRICAL_CABINET".INPUT_BREAKER_QFC40 )
      wire#w1
      Coil( "DB2103_ELECTRICAL_CABINET".QFC40_BREAKER_ALARM )
   END_RUNG
   RUNG wire#powerrail
      Contact( "DB2103_ELECTRICAL_CABINET".QFC40_BREAKER_ALARM )
      I_Contact( "DB2120_MPP_ITC_IPC".RESET_FAULTS )
   END_RUNG wire#w1
   RUNG wire#w1
      Coil( "DB426_ALARMS_WARNINGS".ALARMS.GENERAL."702726" )
   END_RUNG
   // the same network as SCL:
   "DB2103_ELECTRICAL_CABINET".QFC40_BREAKER_ALARM := "DB2103_ELECTRICAL_CABINET".INPUT_BREAKER_QFC40 OR ("DB2103_ELECTRICAL_CABINET".QFC40_BREAKER_ALARM AND NOT "DB2120_MPP_ITC_IPC".RESET_FAULTS);
   "DB426_ALARMS_WARNINGS".ALARMS.GENERAL."702726" := "DB2103_ELECTRICAL_CABINET".QFC40_BREAKER_ALARM;
END_REGION

REGION Network 50: ALARM QB02 CIRCUIT BREAKER TRIPPED
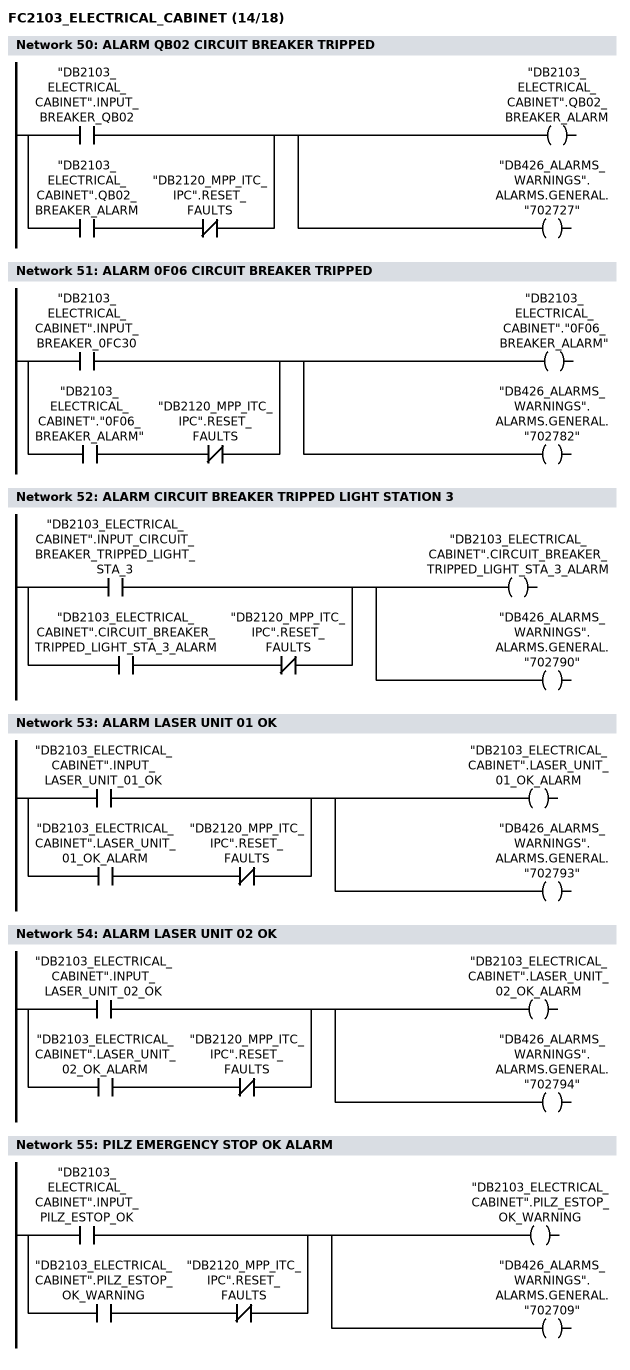
   RUNG wire#powerrail
      Contact( "DB2103_ELECTRICAL_CABINET".INPUT_BREAKER_QB02 )
      wire#w1
      Coil( "DB2103_ELECTRICAL_CABINET".QB02_BREAKER_ALARM )
   END_RUNG
   RUNG wire#powerrail
      Contact( "DB2103_ELECTRICAL_CABINET".QB02_BREAKER_ALARM )
      I_Contact( "DB2120_MPP_ITC_IPC".RESET_FAULTS )
   END_RUNG wire#w1
   RUNG wire#w1
      Coil( "DB426_ALARMS_WARNINGS".ALARMS.GENERAL."702727" )
   END_RUNG
   // the same network as SCL:
   "DB2103_ELECTRICAL_CABINET".QB02_BREAKER_ALARM := "DB2103_ELECTRICAL_CABINET".INPUT_BREAKER_QB02 OR ("DB2103_ELECTRICAL_CABINET".QB02_BREAKER_ALARM AND NOT "DB2120_MPP_ITC_IPC".RESET_FAULTS);
   "DB426_ALARMS_WARNINGS".ALARMS.GENERAL."702727" := "DB2103_ELECTRICAL_CABINET".QB02_BREAKER_ALARM;
END_REGION

REGION Network 51: ALARM 0F06 CIRCUIT BREAKER TRIPPED
   RUNG wire#powerrail
      Contact( "DB2103_ELECTRICAL_CABINET".INPUT_BREAKER_0FC30 )
      wire#w1
      Coil( "DB2103_ELECTRICAL_CABINET"."0F06_BREAKER_ALARM" )
   END_RUNG
   RUNG wire#powerrail
      Contact( "DB2103_ELECTRICAL_CABINET"."0F06_BREAKER_ALARM" )
      I_Contact( "DB2120_MPP_ITC_IPC".RESET_FAULTS )
   END_RUNG wire#w1
   RUNG wire#w1
      Coil( "DB426_ALARMS_WARNINGS".ALARMS.GENERAL."702782" )
   END_RUNG
   // the same network as SCL:
   "DB2103_ELECTRICAL_CABINET"."0F06_BREAKER_ALARM" := "DB2103_ELECTRICAL_CABINET".INPUT_BREAKER_0FC30 OR ("DB2103_ELECTRICAL_CABINET"."0F06_BREAKER_ALARM" AND NOT "DB2120_MPP_ITC_IPC".RESET_FAULTS);
   "DB426_ALARMS_WARNINGS".ALARMS.GENERAL."702782" := "DB2103_ELECTRICAL_CABINET"."0F06_BREAKER_ALARM";
END_REGION

REGION Network 52: ALARM CIRCUIT BREAKER TRIPPED LIGHT STATION 3
   RUNG wire#powerrail
      Contact( "DB2103_ELECTRICAL_CABINET".INPUT_CIRCUIT_BREAKER_TRIPPED_LIGHT_STA_3 )
      wire#w1
      Coil( "DB2103_ELECTRICAL_CABINET".CIRCUIT_BREAKER_TRIPPED_LIGHT_STA_3_ALARM )
   END_RUNG
   RUNG wire#powerrail
      Contact( "DB2103_ELECTRICAL_CABINET".CIRCUIT_BREAKER_TRIPPED_LIGHT_STA_3_ALARM )
      I_Contact( "DB2120_MPP_ITC_IPC".RESET_FAULTS )
   END_RUNG wire#w1
   RUNG wire#w1
      Coil( "DB426_ALARMS_WARNINGS".ALARMS.GENERAL."702790" )
   END_RUNG
   // the same network as SCL:
   "DB2103_ELECTRICAL_CABINET".CIRCUIT_BREAKER_TRIPPED_LIGHT_STA_3_ALARM := "DB2103_ELECTRICAL_CABINET".INPUT_CIRCUIT_BREAKER_TRIPPED_LIGHT_STA_3 OR ("DB2103_ELECTRICAL_CABINET".CIRCUIT_BREAKER_TRIPPED_LIGHT_STA_3_ALARM AND NOT "DB2120_MPP_ITC_IPC".RESET_FAULTS);
   "DB426_ALARMS_WARNINGS".ALARMS.GENERAL."702790" := "DB2103_ELECTRICAL_CABINET".CIRCUIT_BREAKER_TRIPPED_LIGHT_STA_3_ALARM;
END_REGION

REGION Network 53: ALARM LASER UNIT 01 OK
   RUNG wire#powerrail
      Contact( "DB2103_ELECTRICAL_CABINET".INPUT_LASER_UNIT_01_OK )
      wire#w1
      Coil( "DB2103_ELECTRICAL_CABINET".LASER_UNIT_01_OK_ALARM )
   END_RUNG
   RUNG wire#powerrail
      Contact( "DB2103_ELECTRICAL_CABINET".LASER_UNIT_01_OK_ALARM )
      I_Contact( "DB2120_MPP_ITC_IPC".RESET_FAULTS )
   END_RUNG wire#w1
   RUNG wire#w1
      Coil( "DB426_ALARMS_WARNINGS".ALARMS.GENERAL."702793" )
   END_RUNG
   // the same network as SCL:
   "DB2103_ELECTRICAL_CABINET".LASER_UNIT_01_OK_ALARM := "DB2103_ELECTRICAL_CABINET".INPUT_LASER_UNIT_01_OK OR ("DB2103_ELECTRICAL_CABINET".LASER_UNIT_01_OK_ALARM AND NOT "DB2120_MPP_ITC_IPC".RESET_FAULTS);
   "DB426_ALARMS_WARNINGS".ALARMS.GENERAL."702793" := "DB2103_ELECTRICAL_CABINET".LASER_UNIT_01_OK_ALARM;
END_REGION

REGION Network 54: ALARM LASER UNIT 02 OK
   RUNG wire#powerrail
      Contact( "DB2103_ELECTRICAL_CABINET".INPUT_LASER_UNIT_02_OK )
      wire#w1
      Coil( "DB2103_ELECTRICAL_CABINET".LASER_UNIT_02_OK_ALARM )
   END_RUNG
   RUNG wire#powerrail
      Contact( "DB2103_ELECTRICAL_CABINET".LASER_UNIT_02_OK_ALARM )
      I_Contact( "DB2120_MPP_ITC_IPC".RESET_FAULTS )
   END_RUNG wire#w1
   RUNG wire#w1
      Coil( "DB426_ALARMS_WARNINGS".ALARMS.GENERAL."702794" )
   END_RUNG
   // the same network as SCL:
   "DB2103_ELECTRICAL_CABINET".LASER_UNIT_02_OK_ALARM := "DB2103_ELECTRICAL_CABINET".INPUT_LASER_UNIT_02_OK OR ("DB2103_ELECTRICAL_CABINET".LASER_UNIT_02_OK_ALARM AND NOT "DB2120_MPP_ITC_IPC".RESET_FAULTS);
   "DB426_ALARMS_WARNINGS".ALARMS.GENERAL."702794" := "DB2103_ELECTRICAL_CABINET".LASER_UNIT_02_OK_ALARM;
END_REGION

REGION Network 55: PILZ EMERGENCY STOP OK ALARM
   RUNG wire#powerrail
      Contact( "DB2103_ELECTRICAL_CABINET".INPUT_PILZ_ESTOP_OK )
      wire#w1
      Coil( "DB2103_ELECTRICAL_CABINET".PILZ_ESTOP_OK_WARNING )
   END_RUNG
   RUNG wire#powerrail
      Contact( "DB2103_ELECTRICAL_CABINET".PILZ_ESTOP_OK_WARNING )
      I_Contact( "DB2120_MPP_ITC_IPC".RESET_FAULTS )
   END_RUNG wire#w1
   RUNG wire#w1
      Coil( "DB426_ALARMS_WARNINGS".ALARMS.GENERAL."702709" )
   END_RUNG
   // the same network as SCL:
   "DB2103_ELECTRICAL_CABINET".PILZ_ESTOP_OK_WARNING := "DB2103_ELECTRICAL_CABINET".INPUT_PILZ_ESTOP_OK OR ("DB2103_ELECTRICAL_CABINET".PILZ_ESTOP_OK_WARNING AND NOT "DB2120_MPP_ITC_IPC".RESET_FAULTS);
   "DB426_ALARMS_WARNINGS".ALARMS.GENERAL."702709" := "DB2103_ELECTRICAL_CABINET".PILZ_ESTOP_OK_WARNING;
END_REGION

REGION Network 56: IMMEDIATE STOP ALARMS
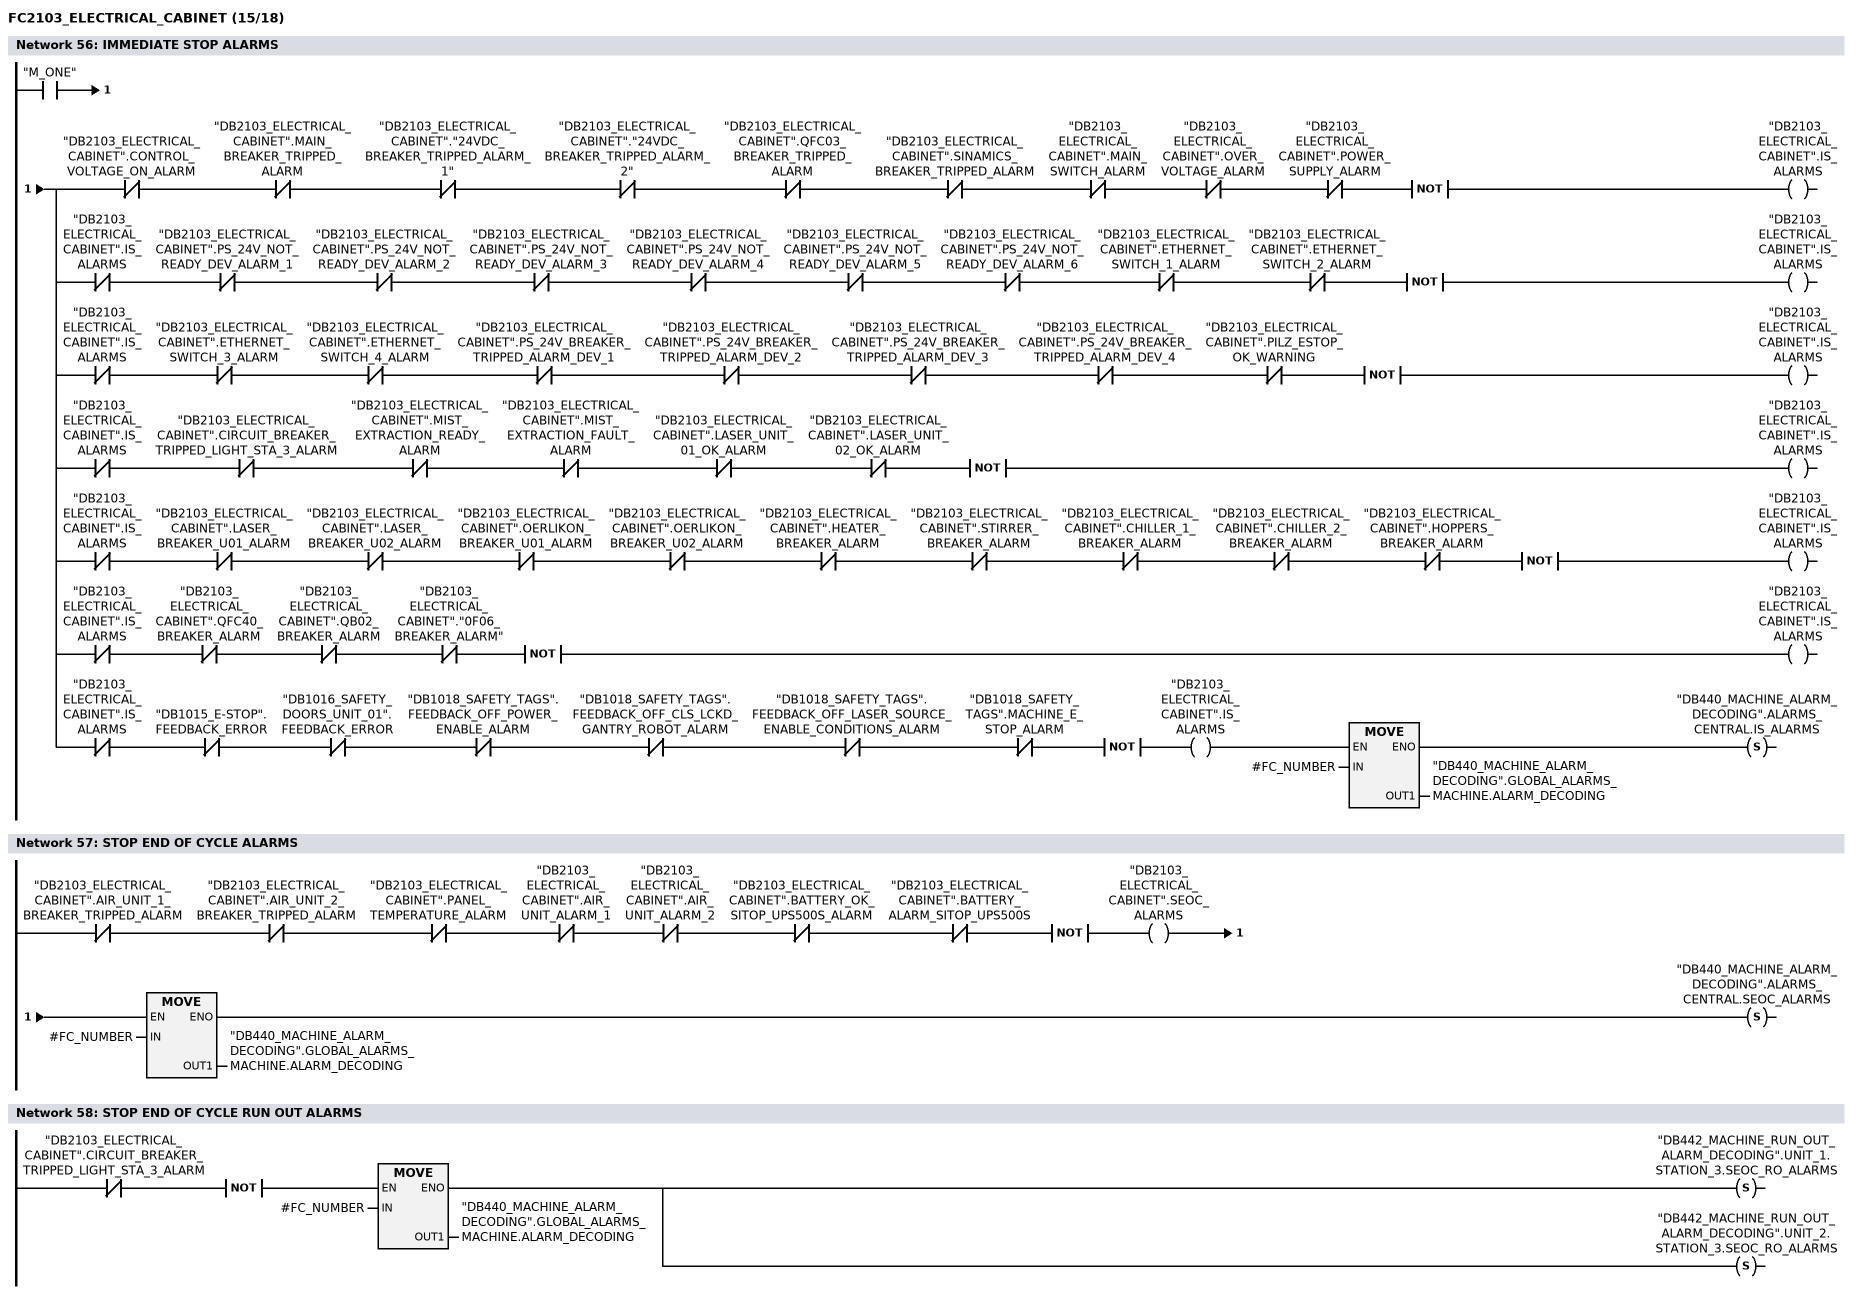
   RUNG wire#powerrail
      Contact( "M_ONE" )
      wire#w1
      I_Contact( "DB2103_ELECTRICAL_CABINET".CONTROL_VOLTAGE_ON_ALARM )
      I_Contact( "DB2103_ELECTRICAL_CABINET".MAIN_BREAKER_TRIPPED_ALARM )
      I_Contact( "DB2103_ELECTRICAL_CABINET"."24VDC_BREAKER_TRIPPED_ALARM_1" )
      I_Contact( "DB2103_ELECTRICAL_CABINET"."24VDC_BREAKER_TRIPPED_ALARM_2" )
      I_Contact( "DB2103_ELECTRICAL_CABINET".QFC03_BREAKER_TRIPPED_ALARM )
      I_Contact( "DB2103_ELECTRICAL_CABINET".SINAMICS_BREAKER_TRIPPED_ALARM )
      I_Contact( "DB2103_ELECTRICAL_CABINET".MAIN_SWITCH_ALARM )
      I_Contact( "DB2103_ELECTRICAL_CABINET".OVER_VOLTAGE_ALARM )
      I_Contact( "DB2103_ELECTRICAL_CABINET".POWER_SUPPLY_ALARM )
      Not()
      Coil( "DB2103_ELECTRICAL_CABINET".IS_ALARMS )
   END_RUNG
   RUNG wire#w1
      I_Contact( "DB2103_ELECTRICAL_CABINET".IS_ALARMS )
      I_Contact( "DB2103_ELECTRICAL_CABINET".PS_24V_NOT_READY_DEV_ALARM_1 )
      I_Contact( "DB2103_ELECTRICAL_CABINET".PS_24V_NOT_READY_DEV_ALARM_2 )
      I_Contact( "DB2103_ELECTRICAL_CABINET".PS_24V_NOT_READY_DEV_ALARM_3 )
      I_Contact( "DB2103_ELECTRICAL_CABINET".PS_24V_NOT_READY_DEV_ALARM_4 )
      I_Contact( "DB2103_ELECTRICAL_CABINET".PS_24V_NOT_READY_DEV_ALARM_5 )
      I_Contact( "DB2103_ELECTRICAL_CABINET".PS_24V_NOT_READY_DEV_ALARM_6 )
      I_Contact( "DB2103_ELECTRICAL_CABINET".ETHERNET_SWITCH_1_ALARM )
      I_Contact( "DB2103_ELECTRICAL_CABINET".ETHERNET_SWITCH_2_ALARM )
      Not()
      Coil( "DB2103_ELECTRICAL_CABINET".IS_ALARMS )
   END_RUNG
   RUNG wire#w1
      I_Contact( "DB2103_ELECTRICAL_CABINET".IS_ALARMS )
      I_Contact( "DB2103_ELECTRICAL_CABINET".ETHERNET_SWITCH_3_ALARM )
      I_Contact( "DB2103_ELECTRICAL_CABINET".ETHERNET_SWITCH_4_ALARM )
      I_Contact( "DB2103_ELECTRICAL_CABINET".PS_24V_BREAKER_TRIPPED_ALARM_DEV_1 )
      I_Contact( "DB2103_ELECTRICAL_CABINET".PS_24V_BREAKER_TRIPPED_ALARM_DEV_2 )
      I_Contact( "DB2103_ELECTRICAL_CABINET".PS_24V_BREAKER_TRIPPED_ALARM_DEV_3 )
      I_Contact( "DB2103_ELECTRICAL_CABINET".PS_24V_BREAKER_TRIPPED_ALARM_DEV_4 )
      I_Contact( "DB2103_ELECTRICAL_CABINET".PILZ_ESTOP_OK_WARNING )
      Not()
      Coil( "DB2103_ELECTRICAL_CABINET".IS_ALARMS )
   END_RUNG
   RUNG wire#w1
      I_Contact( "DB2103_ELECTRICAL_CABINET".IS_ALARMS )
      I_Contact( "DB2103_ELECTRICAL_CABINET".CIRCUIT_BREAKER_TRIPPED_LIGHT_STA_3_ALARM )
      I_Contact( "DB2103_ELECTRICAL_CABINET".MIST_EXTRACTION_READY_ALARM )
      I_Contact( "DB2103_ELECTRICAL_CABINET".MIST_EXTRACTION_FAULT_ALARM )
      I_Contact( "DB2103_ELECTRICAL_CABINET".LASER_UNIT_01_OK_ALARM )
      I_Contact( "DB2103_ELECTRICAL_CABINET".LASER_UNIT_02_OK_ALARM )
      Not()
      Coil( "DB2103_ELECTRICAL_CABINET".IS_ALARMS )
   END_RUNG
   RUNG wire#w1
      I_Contact( "DB2103_ELECTRICAL_CABINET".IS_ALARMS )
      I_Contact( "DB2103_ELECTRICAL_CABINET".LASER_BREAKER_U01_ALARM )
      I_Contact( "DB2103_ELECTRICAL_CABINET".LASER_BREAKER_U02_ALARM )
      I_Contact( "DB2103_ELECTRICAL_CABINET".OERLIKON_BREAKER_U01_ALARM )
      I_Contact( "DB2103_ELECTRICAL_CABINET".OERLIKON_BREAKER_U02_ALARM )
      I_Contact( "DB2103_ELECTRICAL_CABINET".HEATER_BREAKER_ALARM )
      I_Contact( "DB2103_ELECTRICAL_CABINET".STIRRER_BREAKER_ALARM )
      I_Contact( "DB2103_ELECTRICAL_CABINET".CHILLER_1_BREAKER_ALARM )
      I_Contact( "DB2103_ELECTRICAL_CABINET".CHILLER_2_BREAKER_ALARM )
      I_Contact( "DB2103_ELECTRICAL_CABINET".HOPPERS_BREAKER_ALARM )
      Not()
      Coil( "DB2103_ELECTRICAL_CABINET".IS_ALARMS )
   END_RUNG
   RUNG wire#w1
      I_Contact( "DB2103_ELECTRICAL_CABINET".IS_ALARMS )
      I_Contact( "DB2103_ELECTRICAL_CABINET".QFC40_BREAKER_ALARM )
      I_Contact( "DB2103_ELECTRICAL_CABINET".QB02_BREAKER_ALARM )
      I_Contact( "DB2103_ELECTRICAL_CABINET"."0F06_BREAKER_ALARM" )
      Not()
      Coil( "DB2103_ELECTRICAL_CABINET".IS_ALARMS )
   END_RUNG
   RUNG wire#w1
      I_Contact( "DB2103_ELECTRICAL_CABINET".IS_ALARMS )
      I_Contact( "DB1015_E-STOP".FEEDBACK_ERROR )
      I_Contact( "DB1016_SAFETY_DOORS_UNIT_01".FEEDBACK_ERROR )
      I_Contact( "DB1018_SAFETY_TAGS".FEEDBACK_OFF_POWER_ENABLE_ALARM )
      I_Contact( "DB1018_SAFETY_TAGS".FEEDBACK_OFF_CLS_LCKD_GANTRY_ROBOT_ALARM )
      I_Contact( "DB1018_SAFETY_TAGS".FEEDBACK_OFF_LASER_SOURCE_ENABLE_CONDITIONS_ALARM )
      I_Contact( "DB1018_SAFETY_TAGS".MACHINE_E_STOP_ALARM )
      Not()
      Coil( "DB2103_ELECTRICAL_CABINET".IS_ALARMS )
      { S7_GenerateENO := "TRUE" } Move(in := #FC_NUMBER, out1 => "DB440_MACHINE_ALARM_DECODING".GLOBAL_ALARMS_MACHINE.ALARM_DECODING)
      S_Coil( "DB440_MACHINE_ALARM_DECODING".ALARMS_CENTRAL.IS_ALARMS )
   END_RUNG
   // the same network as SCL:
   // ENO of a box is taken as its EN; it also drops when the box reports an error
   "DB2103_ELECTRICAL_CABINET".IS_ALARMS := NOT ("M_ONE" AND NOT "DB2103_ELECTRICAL_CABINET".CONTROL_VOLTAGE_ON_ALARM AND NOT "DB2103_ELECTRICAL_CABINET".MAIN_BREAKER_TRIPPED_ALARM AND NOT "DB2103_ELECTRICAL_CABINET"."24VDC_BREAKER_TRIPPED_ALARM_1" AND NOT "DB2103_ELECTRICAL_CABINET"."24VDC_BREAKER_TRIPPED_ALARM_2" AND NOT "DB2103_ELECTRICAL_CABINET".QFC03_BREAKER_TRIPPED_ALARM AND NOT "DB2103_ELECTRICAL_CABINET".SINAMICS_BREAKER_TRIPPED_ALARM AND NOT "DB2103_ELECTRICAL_CABINET".MAIN_SWITCH_ALARM AND NOT "DB2103_ELECTRICAL_CABINET".OVER_VOLTAGE_ALARM AND NOT "DB2103_ELECTRICAL_CABINET".POWER_SUPPLY_ALARM);
   "DB2103_ELECTRICAL_CABINET".IS_ALARMS := NOT ("M_ONE" AND NOT "DB2103_ELECTRICAL_CABINET".IS_ALARMS AND NOT "DB2103_ELECTRICAL_CABINET".PS_24V_NOT_READY_DEV_ALARM_1 AND NOT "DB2103_ELECTRICAL_CABINET".PS_24V_NOT_READY_DEV_ALARM_2 AND NOT "DB2103_ELECTRICAL_CABINET".PS_24V_NOT_READY_DEV_ALARM_3 AND NOT "DB2103_ELECTRICAL_CABINET".PS_24V_NOT_READY_DEV_ALARM_4 AND NOT "DB2103_ELECTRICAL_CABINET".PS_24V_NOT_READY_DEV_ALARM_5 AND NOT "DB2103_ELECTRICAL_CABINET".PS_24V_NOT_READY_DEV_ALARM_6 AND NOT "DB2103_ELECTRICAL_CABINET".ETHERNET_SWITCH_1_ALARM AND NOT "DB2103_ELECTRICAL_CABINET".ETHERNET_SWITCH_2_ALARM);
   "DB2103_ELECTRICAL_CABINET".IS_ALARMS := NOT ("M_ONE" AND NOT "DB2103_ELECTRICAL_CABINET".IS_ALARMS AND NOT "DB2103_ELECTRICAL_CABINET".ETHERNET_SWITCH_3_ALARM AND NOT "DB2103_ELECTRICAL_CABINET".ETHERNET_SWITCH_4_ALARM AND NOT "DB2103_ELECTRICAL_CABINET".PS_24V_BREAKER_TRIPPED_ALARM_DEV_1 AND NOT "DB2103_ELECTRICAL_CABINET".PS_24V_BREAKER_TRIPPED_ALARM_DEV_2 AND NOT "DB2103_ELECTRICAL_CABINET".PS_24V_BREAKER_TRIPPED_ALARM_DEV_3 AND NOT "DB2103_ELECTRICAL_CABINET".PS_24V_BREAKER_TRIPPED_ALARM_DEV_4 AND NOT "DB2103_ELECTRICAL_CABINET".PILZ_ESTOP_OK_WARNING);
   "DB2103_ELECTRICAL_CABINET".IS_ALARMS := NOT ("M_ONE" AND NOT "DB2103_ELECTRICAL_CABINET".IS_ALARMS AND NOT "DB2103_ELECTRICAL_CABINET".CIRCUIT_BREAKER_TRIPPED_LIGHT_STA_3_ALARM AND NOT "DB2103_ELECTRICAL_CABINET".MIST_EXTRACTION_READY_ALARM AND NOT "DB2103_ELECTRICAL_CABINET".MIST_EXTRACTION_FAULT_ALARM AND NOT "DB2103_ELECTRICAL_CABINET".LASER_UNIT_01_OK_ALARM AND NOT "DB2103_ELECTRICAL_CABINET".LASER_UNIT_02_OK_ALARM);
   "DB2103_ELECTRICAL_CABINET".IS_ALARMS := NOT ("M_ONE" AND NOT "DB2103_ELECTRICAL_CABINET".IS_ALARMS AND NOT "DB2103_ELECTRICAL_CABINET".LASER_BREAKER_U01_ALARM AND NOT "DB2103_ELECTRICAL_CABINET".LASER_BREAKER_U02_ALARM AND NOT "DB2103_ELECTRICAL_CABINET".OERLIKON_BREAKER_U01_ALARM AND NOT "DB2103_ELECTRICAL_CABINET".OERLIKON_BREAKER_U02_ALARM AND NOT "DB2103_ELECTRICAL_CABINET".HEATER_BREAKER_ALARM AND NOT "DB2103_ELECTRICAL_CABINET".STIRRER_BREAKER_ALARM AND NOT "DB2103_ELECTRICAL_CABINET".CHILLER_1_BREAKER_ALARM AND NOT "DB2103_ELECTRICAL_CABINET".CHILLER_2_BREAKER_ALARM AND NOT "DB2103_ELECTRICAL_CABINET".HOPPERS_BREAKER_ALARM);
   "DB2103_ELECTRICAL_CABINET".IS_ALARMS := NOT ("M_ONE" AND NOT "DB2103_ELECTRICAL_CABINET".IS_ALARMS AND NOT "DB2103_ELECTRICAL_CABINET".QFC40_BREAKER_ALARM AND NOT "DB2103_ELECTRICAL_CABINET".QB02_BREAKER_ALARM AND NOT "DB2103_ELECTRICAL_CABINET"."0F06_BREAKER_ALARM");
   "DB2103_ELECTRICAL_CABINET".IS_ALARMS := NOT ("M_ONE" AND NOT "DB2103_ELECTRICAL_CABINET".IS_ALARMS AND NOT "DB1015_E-STOP".FEEDBACK_ERROR AND NOT "DB1016_SAFETY_DOORS_UNIT_01".FEEDBACK_ERROR AND NOT "DB1018_SAFETY_TAGS".FEEDBACK_OFF_POWER_ENABLE_ALARM AND NOT "DB1018_SAFETY_TAGS".FEEDBACK_OFF_CLS_LCKD_GANTRY_ROBOT_ALARM AND NOT "DB1018_SAFETY_TAGS".FEEDBACK_OFF_LASER_SOURCE_ENABLE_CONDITIONS_ALARM AND NOT "DB1018_SAFETY_TAGS".MACHINE_E_STOP_ALARM);
   IF "DB2103_ELECTRICAL_CABINET".IS_ALARMS THEN
       "DB440_MACHINE_ALARM_DECODING".GLOBAL_ALARMS_MACHINE.ALARM_DECODING := #FC_NUMBER;
       "DB440_MACHINE_ALARM_DECODING".ALARMS_CENTRAL.IS_ALARMS := TRUE;
   END_IF;
END_REGION

REGION Network 57: STOP END OF CYCLE ALARMS
   RUNG wire#powerrail
      I_Contact( "DB2103_ELECTRICAL_CABINET".AIR_UNIT_1_BREAKER_TRIPPED_ALARM )
      I_Contact( "DB2103_ELECTRICAL_CABINET".AIR_UNIT_2_BREAKER_TRIPPED_ALARM )
      I_Contact( "DB2103_ELECTRICAL_CABINET".PANEL_TEMPERATURE_ALARM )
      I_Contact( "DB2103_ELECTRICAL_CABINET".AIR_UNIT_ALARM_1 )
      I_Contact( "DB2103_ELECTRICAL_CABINET".AIR_UNIT_ALARM_2 )
      I_Contact( "DB2103_ELECTRICAL_CABINET".BATTERY_OK_SITOP_UPS500S_ALARM )
      I_Contact( "DB2103_ELECTRICAL_CABINET".BATTERY_ALARM_SITOP_UPS500S )
      Not()
      Coil( "DB2103_ELECTRICAL_CABINET".SEOC_ALARMS )
      { S7_GenerateENO := "TRUE" } Move(in := #FC_NUMBER, out1 => "DB440_MACHINE_ALARM_DECODING".GLOBAL_ALARMS_MACHINE.ALARM_DECODING)
      S_Coil( "DB440_MACHINE_ALARM_DECODING".ALARMS_CENTRAL.SEOC_ALARMS )
   END_RUNG
   // the same network as SCL:
   // ENO of a box is taken as its EN; it also drops when the box reports an error
   "DB2103_ELECTRICAL_CABINET".SEOC_ALARMS := NOT (NOT "DB2103_ELECTRICAL_CABINET".AIR_UNIT_1_BREAKER_TRIPPED_ALARM AND NOT "DB2103_ELECTRICAL_CABINET".AIR_UNIT_2_BREAKER_TRIPPED_ALARM AND NOT "DB2103_ELECTRICAL_CABINET".PANEL_TEMPERATURE_ALARM AND NOT "DB2103_ELECTRICAL_CABINET".AIR_UNIT_ALARM_1 AND NOT "DB2103_ELECTRICAL_CABINET".AIR_UNIT_ALARM_2 AND NOT "DB2103_ELECTRICAL_CABINET".BATTERY_OK_SITOP_UPS500S_ALARM AND NOT "DB2103_ELECTRICAL_CABINET".BATTERY_ALARM_SITOP_UPS500S);
   IF "DB2103_ELECTRICAL_CABINET".SEOC_ALARMS THEN
       "DB440_MACHINE_ALARM_DECODING".GLOBAL_ALARMS_MACHINE.ALARM_DECODING := #FC_NUMBER;
       "DB440_MACHINE_ALARM_DECODING".ALARMS_CENTRAL.SEOC_ALARMS := TRUE;
   END_IF;
END_REGION

REGION Network 58: STOP END OF CYCLE RUN OUT ALARMS
   RUNG wire#powerrail
      I_Contact( "DB2103_ELECTRICAL_CABINET".CIRCUIT_BREAKER_TRIPPED_LIGHT_STA_3_ALARM )
      Not()
      Move(in := #FC_NUMBER, out1 => "DB440_MACHINE_ALARM_DECODING".GLOBAL_ALARMS_MACHINE.ALARM_DECODING)
      wire#w1
      S_Coil( "DB442_MACHINE_RUN_OUT_ALARM_DECODING".UNIT_1.STATION_3.SEOC_RO_ALARMS )
   END_RUNG
   RUNG wire#w1
      S_Coil( "DB442_MACHINE_RUN_OUT_ALARM_DECODING".UNIT_2.STATION_3.SEOC_RO_ALARMS )
   END_RUNG
   // the same network as SCL:
   IF NOT (NOT "DB2103_ELECTRICAL_CABINET".CIRCUIT_BREAKER_TRIPPED_LIGHT_STA_3_ALARM) THEN
       "DB440_MACHINE_ALARM_DECODING".GLOBAL_ALARMS_MACHINE.ALARM_DECODING := #FC_NUMBER;
       "DB442_MACHINE_RUN_OUT_ALARM_DECODING".UNIT_1.STATION_3.SEOC_RO_ALARMS := TRUE;
       "DB442_MACHINE_RUN_OUT_ALARM_DECODING".UNIT_2.STATION_3.SEOC_RO_ALARMS := TRUE;
   END_IF;
END_REGION

REGION Network 59: PROGRESSIVE STOP POWDER ALARMS
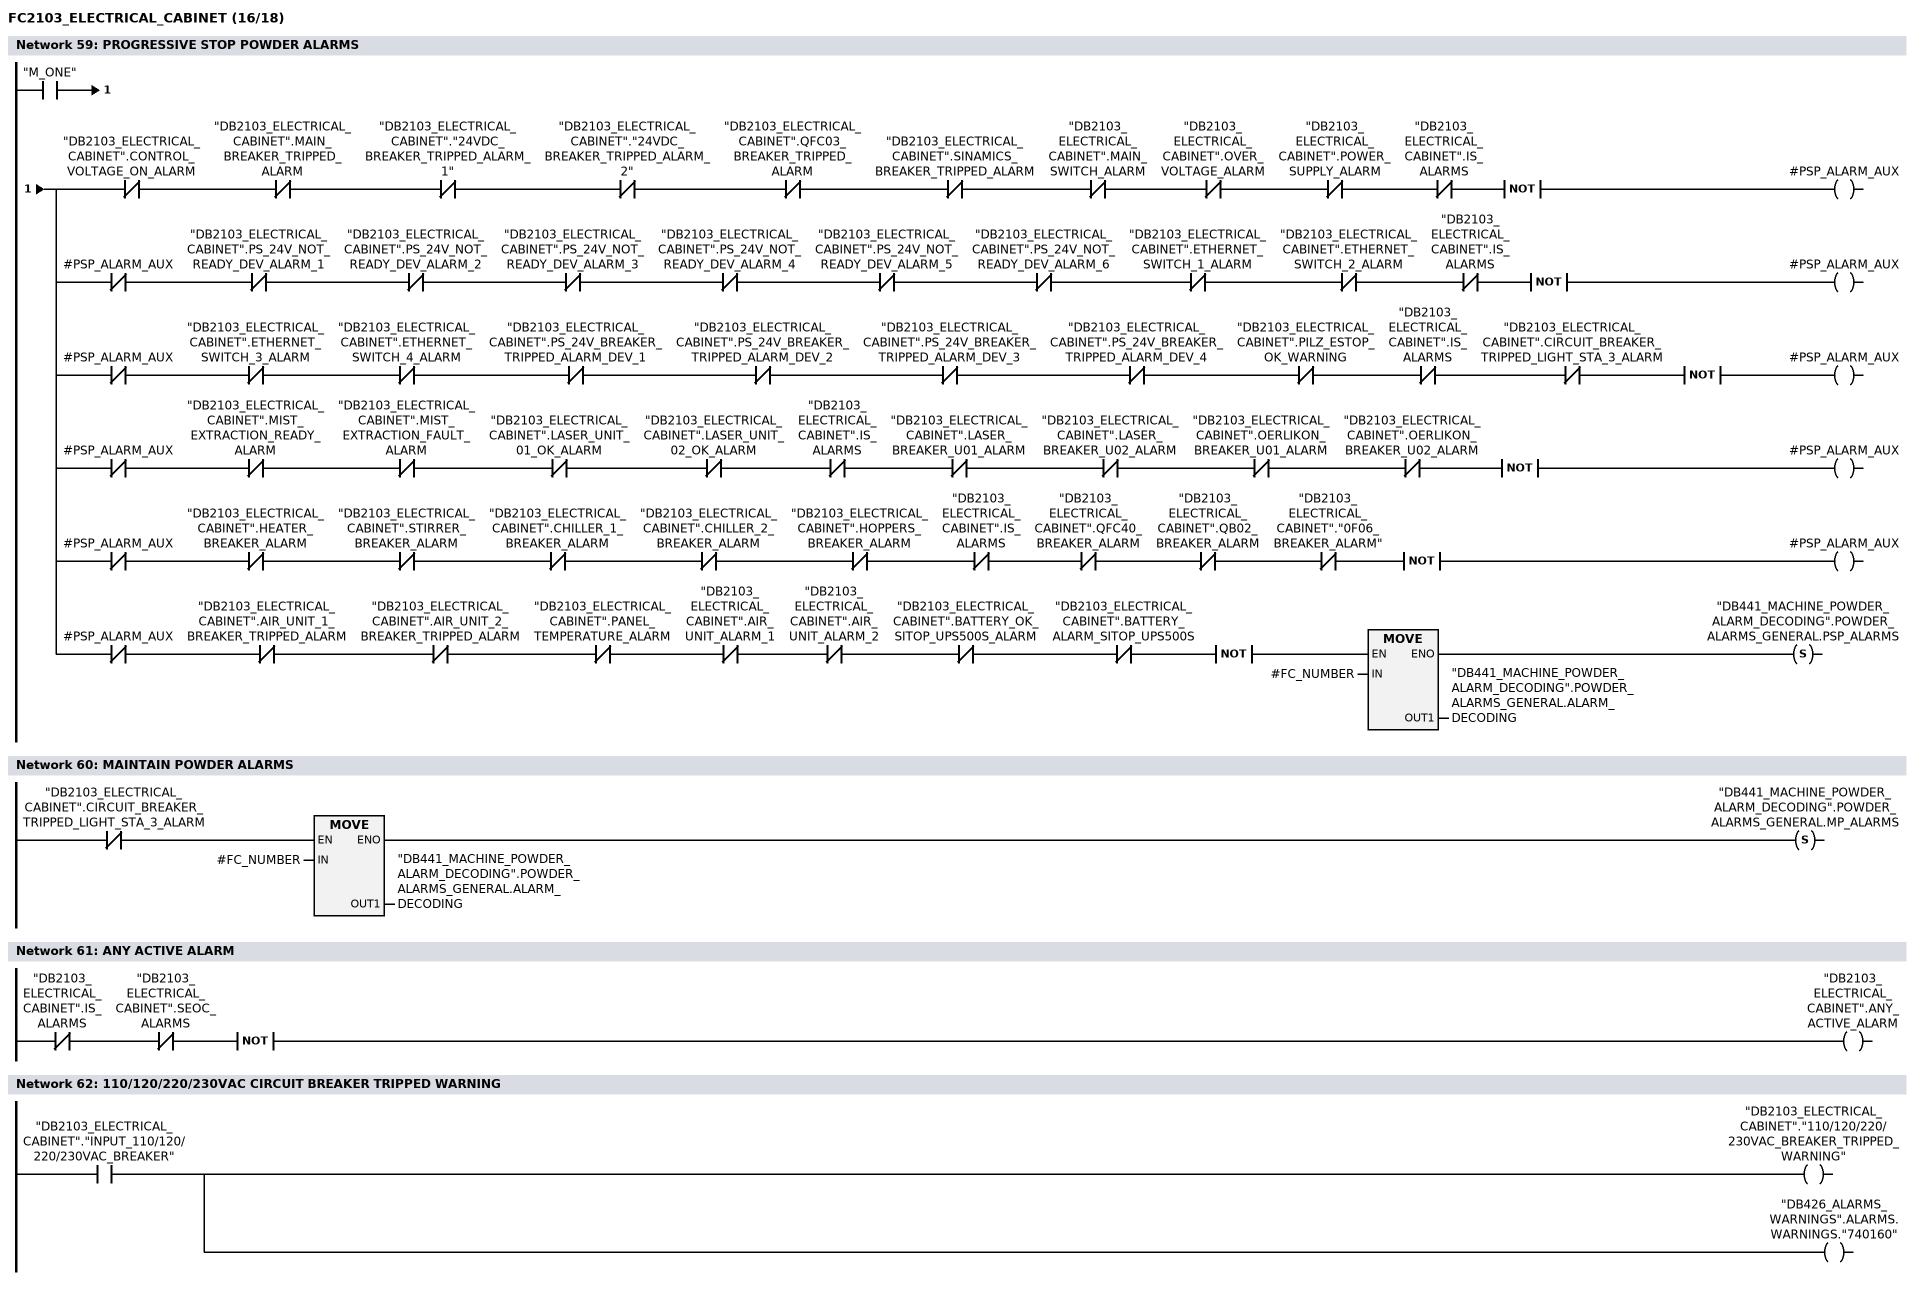
   RUNG wire#powerrail
      Contact( "M_ONE" )
      wire#w1
      I_Contact( "DB2103_ELECTRICAL_CABINET".CONTROL_VOLTAGE_ON_ALARM )
      I_Contact( "DB2103_ELECTRICAL_CABINET".MAIN_BREAKER_TRIPPED_ALARM )
      I_Contact( "DB2103_ELECTRICAL_CABINET"."24VDC_BREAKER_TRIPPED_ALARM_1" )
      I_Contact( "DB2103_ELECTRICAL_CABINET"."24VDC_BREAKER_TRIPPED_ALARM_2" )
      I_Contact( "DB2103_ELECTRICAL_CABINET".QFC03_BREAKER_TRIPPED_ALARM )
      I_Contact( "DB2103_ELECTRICAL_CABINET".SINAMICS_BREAKER_TRIPPED_ALARM )
      I_Contact( "DB2103_ELECTRICAL_CABINET".MAIN_SWITCH_ALARM )
      I_Contact( "DB2103_ELECTRICAL_CABINET".OVER_VOLTAGE_ALARM )
      I_Contact( "DB2103_ELECTRICAL_CABINET".POWER_SUPPLY_ALARM )
      I_Contact( "DB2103_ELECTRICAL_CABINET".IS_ALARMS )
      Not()
      Coil( #PSP_ALARM_AUX )
   END_RUNG
   RUNG wire#w1
      I_Contact( #PSP_ALARM_AUX )
      I_Contact( "DB2103_ELECTRICAL_CABINET".PS_24V_NOT_READY_DEV_ALARM_1 )
      I_Contact( "DB2103_ELECTRICAL_CABINET".PS_24V_NOT_READY_DEV_ALARM_2 )
      I_Contact( "DB2103_ELECTRICAL_CABINET".PS_24V_NOT_READY_DEV_ALARM_3 )
      I_Contact( "DB2103_ELECTRICAL_CABINET".PS_24V_NOT_READY_DEV_ALARM_4 )
      I_Contact( "DB2103_ELECTRICAL_CABINET".PS_24V_NOT_READY_DEV_ALARM_5 )
      I_Contact( "DB2103_ELECTRICAL_CABINET".PS_24V_NOT_READY_DEV_ALARM_6 )
      I_Contact( "DB2103_ELECTRICAL_CABINET".ETHERNET_SWITCH_1_ALARM )
      I_Contact( "DB2103_ELECTRICAL_CABINET".ETHERNET_SWITCH_2_ALARM )
      I_Contact( "DB2103_ELECTRICAL_CABINET".IS_ALARMS )
      Not()
      Coil( #PSP_ALARM_AUX )
   END_RUNG
   RUNG wire#w1
      I_Contact( #PSP_ALARM_AUX )
      I_Contact( "DB2103_ELECTRICAL_CABINET".ETHERNET_SWITCH_3_ALARM )
      I_Contact( "DB2103_ELECTRICAL_CABINET".ETHERNET_SWITCH_4_ALARM )
      I_Contact( "DB2103_ELECTRICAL_CABINET".PS_24V_BREAKER_TRIPPED_ALARM_DEV_1 )
      I_Contact( "DB2103_ELECTRICAL_CABINET".PS_24V_BREAKER_TRIPPED_ALARM_DEV_2 )
      I_Contact( "DB2103_ELECTRICAL_CABINET".PS_24V_BREAKER_TRIPPED_ALARM_DEV_3 )
      I_Contact( "DB2103_ELECTRICAL_CABINET".PS_24V_BREAKER_TRIPPED_ALARM_DEV_4 )
      I_Contact( "DB2103_ELECTRICAL_CABINET".PILZ_ESTOP_OK_WARNING )
      I_Contact( "DB2103_ELECTRICAL_CABINET".IS_ALARMS )
      I_Contact( "DB2103_ELECTRICAL_CABINET".CIRCUIT_BREAKER_TRIPPED_LIGHT_STA_3_ALARM )
      Not()
      Coil( #PSP_ALARM_AUX )
   END_RUNG
   RUNG wire#w1
      I_Contact( #PSP_ALARM_AUX )
      I_Contact( "DB2103_ELECTRICAL_CABINET".MIST_EXTRACTION_READY_ALARM )
      I_Contact( "DB2103_ELECTRICAL_CABINET".MIST_EXTRACTION_FAULT_ALARM )
      I_Contact( "DB2103_ELECTRICAL_CABINET".LASER_UNIT_01_OK_ALARM )
      I_Contact( "DB2103_ELECTRICAL_CABINET".LASER_UNIT_02_OK_ALARM )
      I_Contact( "DB2103_ELECTRICAL_CABINET".IS_ALARMS )
      I_Contact( "DB2103_ELECTRICAL_CABINET".LASER_BREAKER_U01_ALARM )
      I_Contact( "DB2103_ELECTRICAL_CABINET".LASER_BREAKER_U02_ALARM )
      I_Contact( "DB2103_ELECTRICAL_CABINET".OERLIKON_BREAKER_U01_ALARM )
      I_Contact( "DB2103_ELECTRICAL_CABINET".OERLIKON_BREAKER_U02_ALARM )
      Not()
      Coil( #PSP_ALARM_AUX )
   END_RUNG
   RUNG wire#w1
      I_Contact( #PSP_ALARM_AUX )
      I_Contact( "DB2103_ELECTRICAL_CABINET".HEATER_BREAKER_ALARM )
      I_Contact( "DB2103_ELECTRICAL_CABINET".STIRRER_BREAKER_ALARM )
      I_Contact( "DB2103_ELECTRICAL_CABINET".CHILLER_1_BREAKER_ALARM )
      I_Contact( "DB2103_ELECTRICAL_CABINET".CHILLER_2_BREAKER_ALARM )
      I_Contact( "DB2103_ELECTRICAL_CABINET".HOPPERS_BREAKER_ALARM )
      I_Contact( "DB2103_ELECTRICAL_CABINET".IS_ALARMS )
      I_Contact( "DB2103_ELECTRICAL_CABINET".QFC40_BREAKER_ALARM )
      I_Contact( "DB2103_ELECTRICAL_CABINET".QB02_BREAKER_ALARM )
      I_Contact( "DB2103_ELECTRICAL_CABINET"."0F06_BREAKER_ALARM" )
      Not()
      Coil( #PSP_ALARM_AUX )
   END_RUNG
   RUNG wire#w1
      I_Contact( #PSP_ALARM_AUX )
      I_Contact( "DB2103_ELECTRICAL_CABINET".AIR_UNIT_1_BREAKER_TRIPPED_ALARM )
      I_Contact( "DB2103_ELECTRICAL_CABINET".AIR_UNIT_2_BREAKER_TRIPPED_ALARM )
      I_Contact( "DB2103_ELECTRICAL_CABINET".PANEL_TEMPERATURE_ALARM )
      I_Contact( "DB2103_ELECTRICAL_CABINET".AIR_UNIT_ALARM_1 )
      I_Contact( "DB2103_ELECTRICAL_CABINET".AIR_UNIT_ALARM_2 )
      I_Contact( "DB2103_ELECTRICAL_CABINET".BATTERY_OK_SITOP_UPS500S_ALARM )
      I_Contact( "DB2103_ELECTRICAL_CABINET".BATTERY_ALARM_SITOP_UPS500S )
      Not()
      Move(in := #FC_NUMBER, out1 => "DB441_MACHINE_POWDER_ALARM_DECODING".POWDER_ALARMS_GENERAL.ALARM_DECODING)
      S_Coil( "DB441_MACHINE_POWDER_ALARM_DECODING".POWDER_ALARMS_GENERAL.PSP_ALARMS )
   END_RUNG
   // the same network as SCL:
   #PSP_ALARM_AUX := NOT ("M_ONE" AND NOT "DB2103_ELECTRICAL_CABINET".CONTROL_VOLTAGE_ON_ALARM AND NOT "DB2103_ELECTRICAL_CABINET".MAIN_BREAKER_TRIPPED_ALARM AND NOT "DB2103_ELECTRICAL_CABINET"."24VDC_BREAKER_TRIPPED_ALARM_1" AND NOT "DB2103_ELECTRICAL_CABINET"."24VDC_BREAKER_TRIPPED_ALARM_2" AND NOT "DB2103_ELECTRICAL_CABINET".QFC03_BREAKER_TRIPPED_ALARM AND NOT "DB2103_ELECTRICAL_CABINET".SINAMICS_BREAKER_TRIPPED_ALARM AND NOT "DB2103_ELECTRICAL_CABINET".MAIN_SWITCH_ALARM AND NOT "DB2103_ELECTRICAL_CABINET".OVER_VOLTAGE_ALARM AND NOT "DB2103_ELECTRICAL_CABINET".POWER_SUPPLY_ALARM AND NOT "DB2103_ELECTRICAL_CABINET".IS_ALARMS);
   #PSP_ALARM_AUX := NOT ("M_ONE" AND NOT #PSP_ALARM_AUX AND NOT "DB2103_ELECTRICAL_CABINET".PS_24V_NOT_READY_DEV_ALARM_1 AND NOT "DB2103_ELECTRICAL_CABINET".PS_24V_NOT_READY_DEV_ALARM_2 AND NOT "DB2103_ELECTRICAL_CABINET".PS_24V_NOT_READY_DEV_ALARM_3 AND NOT "DB2103_ELECTRICAL_CABINET".PS_24V_NOT_READY_DEV_ALARM_4 AND NOT "DB2103_ELECTRICAL_CABINET".PS_24V_NOT_READY_DEV_ALARM_5 AND NOT "DB2103_ELECTRICAL_CABINET".PS_24V_NOT_READY_DEV_ALARM_6 AND NOT "DB2103_ELECTRICAL_CABINET".ETHERNET_SWITCH_1_ALARM AND NOT "DB2103_ELECTRICAL_CABINET".ETHERNET_SWITCH_2_ALARM AND NOT "DB2103_ELECTRICAL_CABINET".IS_ALARMS);
   #PSP_ALARM_AUX := NOT ("M_ONE" AND NOT #PSP_ALARM_AUX AND NOT "DB2103_ELECTRICAL_CABINET".ETHERNET_SWITCH_3_ALARM AND NOT "DB2103_ELECTRICAL_CABINET".ETHERNET_SWITCH_4_ALARM AND NOT "DB2103_ELECTRICAL_CABINET".PS_24V_BREAKER_TRIPPED_ALARM_DEV_1 AND NOT "DB2103_ELECTRICAL_CABINET".PS_24V_BREAKER_TRIPPED_ALARM_DEV_2 AND NOT "DB2103_ELECTRICAL_CABINET".PS_24V_BREAKER_TRIPPED_ALARM_DEV_3 AND NOT "DB2103_ELECTRICAL_CABINET".PS_24V_BREAKER_TRIPPED_ALARM_DEV_4 AND NOT "DB2103_ELECTRICAL_CABINET".PILZ_ESTOP_OK_WARNING AND NOT "DB2103_ELECTRICAL_CABINET".IS_ALARMS AND NOT "DB2103_ELECTRICAL_CABINET".CIRCUIT_BREAKER_TRIPPED_LIGHT_STA_3_ALARM);
   #PSP_ALARM_AUX := NOT ("M_ONE" AND NOT #PSP_ALARM_AUX AND NOT "DB2103_ELECTRICAL_CABINET".MIST_EXTRACTION_READY_ALARM AND NOT "DB2103_ELECTRICAL_CABINET".MIST_EXTRACTION_FAULT_ALARM AND NOT "DB2103_ELECTRICAL_CABINET".LASER_UNIT_01_OK_ALARM AND NOT "DB2103_ELECTRICAL_CABINET".LASER_UNIT_02_OK_ALARM AND NOT "DB2103_ELECTRICAL_CABINET".IS_ALARMS AND NOT "DB2103_ELECTRICAL_CABINET".LASER_BREAKER_U01_ALARM AND NOT "DB2103_ELECTRICAL_CABINET".LASER_BREAKER_U02_ALARM AND NOT "DB2103_ELECTRICAL_CABINET".OERLIKON_BREAKER_U01_ALARM AND NOT "DB2103_ELECTRICAL_CABINET".OERLIKON_BREAKER_U02_ALARM);
   #PSP_ALARM_AUX := NOT ("M_ONE" AND NOT #PSP_ALARM_AUX AND NOT "DB2103_ELECTRICAL_CABINET".HEATER_BREAKER_ALARM AND NOT "DB2103_ELECTRICAL_CABINET".STIRRER_BREAKER_ALARM AND NOT "DB2103_ELECTRICAL_CABINET".CHILLER_1_BREAKER_ALARM AND NOT "DB2103_ELECTRICAL_CABINET".CHILLER_2_BREAKER_ALARM AND NOT "DB2103_ELECTRICAL_CABINET".HOPPERS_BREAKER_ALARM AND NOT "DB2103_ELECTRICAL_CABINET".IS_ALARMS AND NOT "DB2103_ELECTRICAL_CABINET".QFC40_BREAKER_ALARM AND NOT "DB2103_ELECTRICAL_CABINET".QB02_BREAKER_ALARM AND NOT "DB2103_ELECTRICAL_CABINET"."0F06_BREAKER_ALARM");
   IF NOT ("M_ONE" AND NOT #PSP_ALARM_AUX AND NOT "DB2103_ELECTRICAL_CABINET".AIR_UNIT_1_BREAKER_TRIPPED_ALARM AND NOT "DB2103_ELECTRICAL_CABINET".AIR_UNIT_2_BREAKER_TRIPPED_ALARM AND NOT "DB2103_ELECTRICAL_CABINET".PANEL_TEMPERATURE_ALARM AND NOT "DB2103_ELECTRICAL_CABINET".AIR_UNIT_ALARM_1 AND NOT "DB2103_ELECTRICAL_CABINET".AIR_UNIT_ALARM_2 AND NOT "DB2103_ELECTRICAL_CABINET".BATTERY_OK_SITOP_UPS500S_ALARM AND NOT "DB2103_ELECTRICAL_CABINET".BATTERY_ALARM_SITOP_UPS500S) THEN
       "DB441_MACHINE_POWDER_ALARM_DECODING".POWDER_ALARMS_GENERAL.ALARM_DECODING := #FC_NUMBER;
       "DB441_MACHINE_POWDER_ALARM_DECODING".POWDER_ALARMS_GENERAL.PSP_ALARMS := TRUE;
   END_IF;
END_REGION

REGION Network 60: MAINTAIN POWDER ALARMS
   RUNG wire#powerrail
      I_Contact( "DB2103_ELECTRICAL_CABINET".CIRCUIT_BREAKER_TRIPPED_LIGHT_STA_3_ALARM )
      Move(in := #FC_NUMBER, out1 => "DB441_MACHINE_POWDER_ALARM_DECODING".POWDER_ALARMS_GENERAL.ALARM_DECODING)
      S_Coil( "DB441_MACHINE_POWDER_ALARM_DECODING".POWDER_ALARMS_GENERAL.MP_ALARMS )
   END_RUNG
   // the same network as SCL:
   IF NOT "DB2103_ELECTRICAL_CABINET".CIRCUIT_BREAKER_TRIPPED_LIGHT_STA_3_ALARM THEN
       "DB441_MACHINE_POWDER_ALARM_DECODING".POWDER_ALARMS_GENERAL.ALARM_DECODING := #FC_NUMBER;
       "DB441_MACHINE_POWDER_ALARM_DECODING".POWDER_ALARMS_GENERAL.MP_ALARMS := TRUE;
   END_IF;
END_REGION

REGION Network 61: ANY ACTIVE ALARM
   RUNG wire#powerrail
      I_Contact( "DB2103_ELECTRICAL_CABINET".IS_ALARMS )
      I_Contact( "DB2103_ELECTRICAL_CABINET".SEOC_ALARMS )
      Not()
      Coil( "DB2103_ELECTRICAL_CABINET".ANY_ACTIVE_ALARM )
   END_RUNG
   // the same network as SCL:
   "DB2103_ELECTRICAL_CABINET".ANY_ACTIVE_ALARM := NOT (NOT "DB2103_ELECTRICAL_CABINET".IS_ALARMS AND NOT "DB2103_ELECTRICAL_CABINET".SEOC_ALARMS);
END_REGION

REGION Network 62: 110/120/220/230VAC CIRCUIT BREAKER TRIPPED WARNING
   RUNG wire#powerrail
      Contact( "DB2103_ELECTRICAL_CABINET"."INPUT_110/120/220/230VAC_BREAKER" )
      wire#w1
      Coil( "DB2103_ELECTRICAL_CABINET"."110/120/220/230VAC_BREAKER_TRIPPED_WARNING" )
   END_RUNG
   RUNG wire#w1
      Coil( "DB426_ALARMS_WARNINGS".ALARMS.WARNINGS."740160" )
   END_RUNG
   // the same network as SCL:
   "DB2103_ELECTRICAL_CABINET"."110/120/220/230VAC_BREAKER_TRIPPED_WARNING" := "DB2103_ELECTRICAL_CABINET"."INPUT_110/120/220/230VAC_BREAKER";
   "DB426_ALARMS_WARNINGS".ALARMS.WARNINGS."740160" := "DB2103_ELECTRICAL_CABINET"."INPUT_110/120/220/230VAC_BREAKER";
END_REGION

REGION Network 63: CABINET LIGHT CIRCUIT BREAKER TRIPPED WARNING
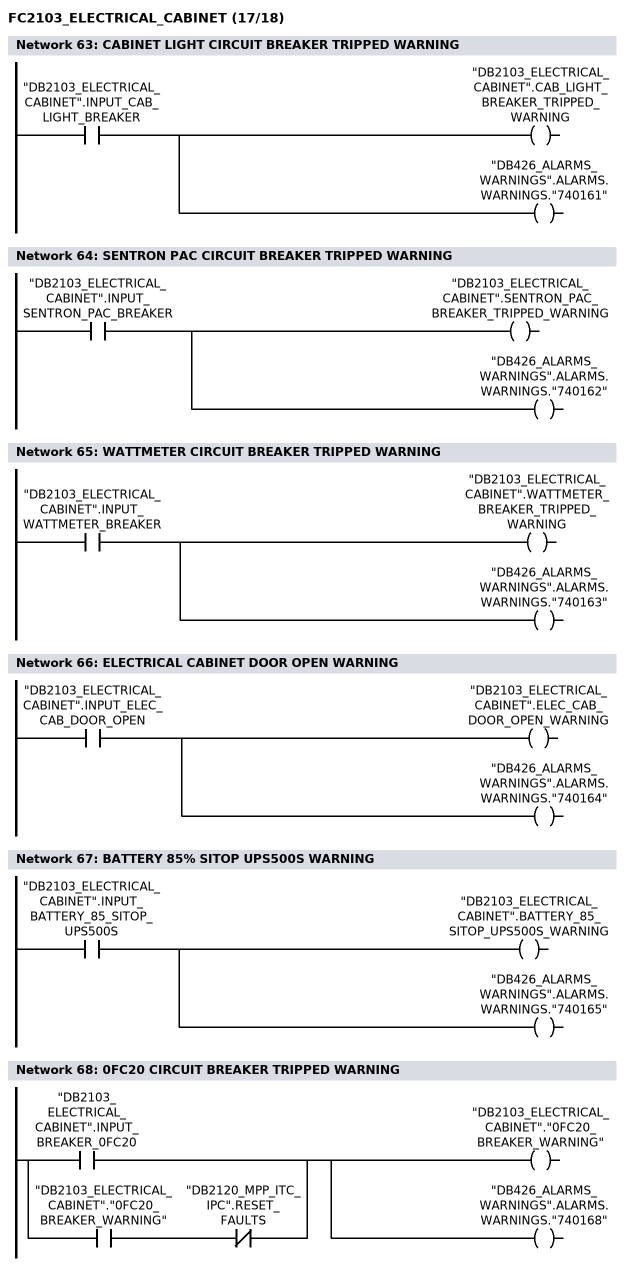
   RUNG wire#powerrail
      Contact( "DB2103_ELECTRICAL_CABINET".INPUT_CAB_LIGHT_BREAKER )
      wire#w1
      Coil( "DB2103_ELECTRICAL_CABINET".CAB_LIGHT_BREAKER_TRIPPED_WARNING )
   END_RUNG
   RUNG wire#w1
      Coil( "DB426_ALARMS_WARNINGS".ALARMS.WARNINGS."740161" )
   END_RUNG
   // the same network as SCL:
   "DB2103_ELECTRICAL_CABINET".CAB_LIGHT_BREAKER_TRIPPED_WARNING := "DB2103_ELECTRICAL_CABINET".INPUT_CAB_LIGHT_BREAKER;
   "DB426_ALARMS_WARNINGS".ALARMS.WARNINGS."740161" := "DB2103_ELECTRICAL_CABINET".INPUT_CAB_LIGHT_BREAKER;
END_REGION

REGION Network 64: SENTRON PAC CIRCUIT BREAKER TRIPPED WARNING
   RUNG wire#powerrail
      Contact( "DB2103_ELECTRICAL_CABINET".INPUT_SENTRON_PAC_BREAKER )
      wire#w1
      Coil( "DB2103_ELECTRICAL_CABINET".SENTRON_PAC_BREAKER_TRIPPED_WARNING )
   END_RUNG
   RUNG wire#w1
      Coil( "DB426_ALARMS_WARNINGS".ALARMS.WARNINGS."740162" )
   END_RUNG
   // the same network as SCL:
   "DB2103_ELECTRICAL_CABINET".SENTRON_PAC_BREAKER_TRIPPED_WARNING := "DB2103_ELECTRICAL_CABINET".INPUT_SENTRON_PAC_BREAKER;
   "DB426_ALARMS_WARNINGS".ALARMS.WARNINGS."740162" := "DB2103_ELECTRICAL_CABINET".INPUT_SENTRON_PAC_BREAKER;
END_REGION

REGION Network 65: WATTMETER CIRCUIT BREAKER TRIPPED WARNING
   RUNG wire#powerrail
      Contact( "DB2103_ELECTRICAL_CABINET".INPUT_WATTMETER_BREAKER )
      wire#w1
      Coil( "DB2103_ELECTRICAL_CABINET".WATTMETER_BREAKER_TRIPPED_WARNING )
   END_RUNG
   RUNG wire#w1
      Coil( "DB426_ALARMS_WARNINGS".ALARMS.WARNINGS."740163" )
   END_RUNG
   // the same network as SCL:
   "DB2103_ELECTRICAL_CABINET".WATTMETER_BREAKER_TRIPPED_WARNING := "DB2103_ELECTRICAL_CABINET".INPUT_WATTMETER_BREAKER;
   "DB426_ALARMS_WARNINGS".ALARMS.WARNINGS."740163" := "DB2103_ELECTRICAL_CABINET".INPUT_WATTMETER_BREAKER;
END_REGION

REGION Network 66: ELECTRICAL CABINET DOOR OPEN WARNING
   RUNG wire#powerrail
      Contact( "DB2103_ELECTRICAL_CABINET".INPUT_ELEC_CAB_DOOR_OPEN )
      wire#w1
      Coil( "DB2103_ELECTRICAL_CABINET".ELEC_CAB_DOOR_OPEN_WARNING )
   END_RUNG
   RUNG wire#w1
      Coil( "DB426_ALARMS_WARNINGS".ALARMS.WARNINGS."740164" )
   END_RUNG
   // the same network as SCL:
   "DB2103_ELECTRICAL_CABINET".ELEC_CAB_DOOR_OPEN_WARNING := "DB2103_ELECTRICAL_CABINET".INPUT_ELEC_CAB_DOOR_OPEN;
   "DB426_ALARMS_WARNINGS".ALARMS.WARNINGS."740164" := "DB2103_ELECTRICAL_CABINET".INPUT_ELEC_CAB_DOOR_OPEN;
END_REGION

REGION Network 67: BATTERY 85% SITOP UPS500S WARNING
   RUNG wire#powerrail
      Contact( "DB2103_ELECTRICAL_CABINET".INPUT_BATTERY_85_SITOP_UPS500S )
      wire#w1
      Coil( "DB2103_ELECTRICAL_CABINET".BATTERY_85_SITOP_UPS500S_WARNING )
   END_RUNG
   RUNG wire#w1
      Coil( "DB426_ALARMS_WARNINGS".ALARMS.WARNINGS."740165" )
   END_RUNG
   // the same network as SCL:
   "DB2103_ELECTRICAL_CABINET".BATTERY_85_SITOP_UPS500S_WARNING := "DB2103_ELECTRICAL_CABINET".INPUT_BATTERY_85_SITOP_UPS500S;
   "DB426_ALARMS_WARNINGS".ALARMS.WARNINGS."740165" := "DB2103_ELECTRICAL_CABINET".INPUT_BATTERY_85_SITOP_UPS500S;
END_REGION

REGION Network 68: 0FC20 CIRCUIT BREAKER TRIPPED WARNING
   RUNG wire#powerrail
      Contact( "DB2103_ELECTRICAL_CABINET".INPUT_BREAKER_0FC20 )
      wire#w1
      Coil( "DB2103_ELECTRICAL_CABINET"."0FC20_BREAKER_WARNING" )
   END_RUNG
   RUNG wire#powerrail
      Contact( "DB2103_ELECTRICAL_CABINET"."0FC20_BREAKER_WARNING" )
      I_Contact( "DB2120_MPP_ITC_IPC".RESET_FAULTS )
   END_RUNG wire#w1
   RUNG wire#w1
      Coil( "DB426_ALARMS_WARNINGS".ALARMS.WARNINGS."740168" )
   END_RUNG
   // the same network as SCL:
   "DB2103_ELECTRICAL_CABINET"."0FC20_BREAKER_WARNING" := "DB2103_ELECTRICAL_CABINET".INPUT_BREAKER_0FC20 OR ("DB2103_ELECTRICAL_CABINET"."0FC20_BREAKER_WARNING" AND NOT "DB2120_MPP_ITC_IPC".RESET_FAULTS);
   "DB426_ALARMS_WARNINGS".ALARMS.WARNINGS."740168" := "DB2103_ELECTRICAL_CABINET"."0FC20_BREAKER_WARNING";
END_REGION

REGION Network 69: 0FC21 CIRCUIT BREAKER TRIPPED WARNING
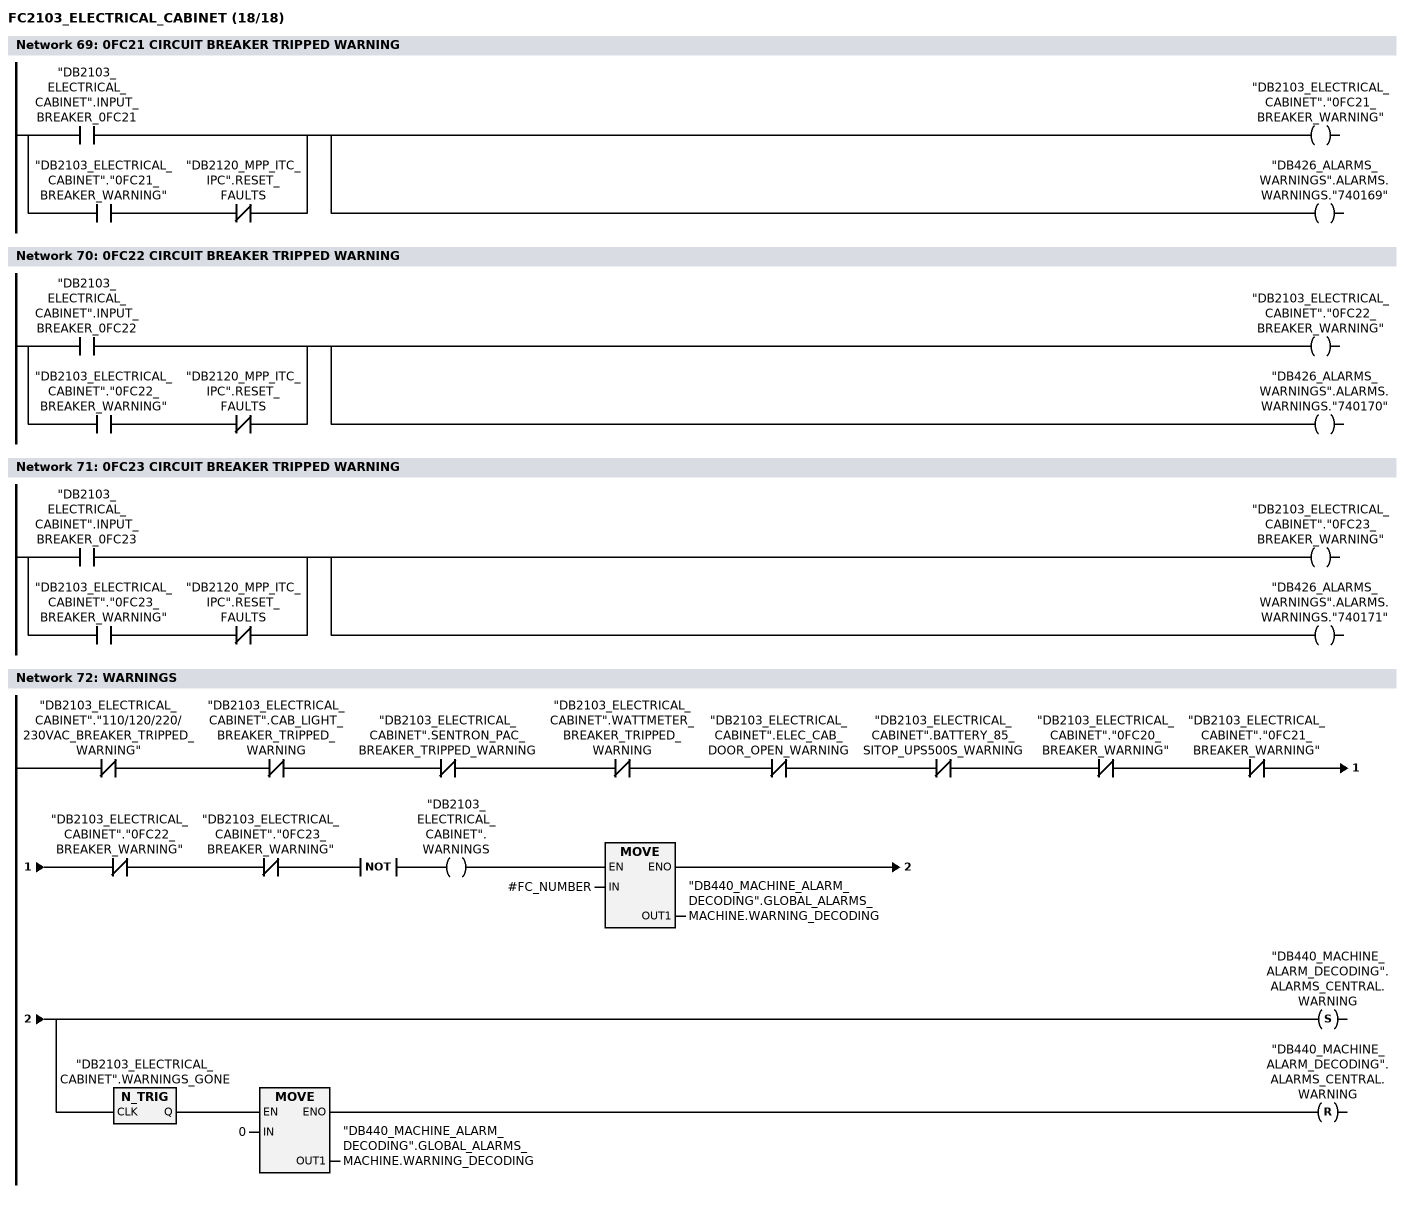
   RUNG wire#powerrail
      Contact( "DB2103_ELECTRICAL_CABINET".INPUT_BREAKER_0FC21 )
      wire#w1
      Coil( "DB2103_ELECTRICAL_CABINET"."0FC21_BREAKER_WARNING" )
   END_RUNG
   RUNG wire#powerrail
      Contact( "DB2103_ELECTRICAL_CABINET"."0FC21_BREAKER_WARNING" )
      I_Contact( "DB2120_MPP_ITC_IPC".RESET_FAULTS )
   END_RUNG wire#w1
   RUNG wire#w1
      Coil( "DB426_ALARMS_WARNINGS".ALARMS.WARNINGS."740169" )
   END_RUNG
   // the same network as SCL:
   "DB2103_ELECTRICAL_CABINET"."0FC21_BREAKER_WARNING" := "DB2103_ELECTRICAL_CABINET".INPUT_BREAKER_0FC21 OR ("DB2103_ELECTRICAL_CABINET"."0FC21_BREAKER_WARNING" AND NOT "DB2120_MPP_ITC_IPC".RESET_FAULTS);
   "DB426_ALARMS_WARNINGS".ALARMS.WARNINGS."740169" := "DB2103_ELECTRICAL_CABINET"."0FC21_BREAKER_WARNING";
END_REGION

REGION Network 70: 0FC22 CIRCUIT BREAKER TRIPPED WARNING
   RUNG wire#powerrail
      Contact( "DB2103_ELECTRICAL_CABINET".INPUT_BREAKER_0FC22 )
      wire#w1
      Coil( "DB2103_ELECTRICAL_CABINET"."0FC22_BREAKER_WARNING" )
   END_RUNG
   RUNG wire#powerrail
      Contact( "DB2103_ELECTRICAL_CABINET"."0FC22_BREAKER_WARNING" )
      I_Contact( "DB2120_MPP_ITC_IPC".RESET_FAULTS )
   END_RUNG wire#w1
   RUNG wire#w1
      Coil( "DB426_ALARMS_WARNINGS".ALARMS.WARNINGS."740170" )
   END_RUNG
   // the same network as SCL:
   "DB2103_ELECTRICAL_CABINET"."0FC22_BREAKER_WARNING" := "DB2103_ELECTRICAL_CABINET".INPUT_BREAKER_0FC22 OR ("DB2103_ELECTRICAL_CABINET"."0FC22_BREAKER_WARNING" AND NOT "DB2120_MPP_ITC_IPC".RESET_FAULTS);
   "DB426_ALARMS_WARNINGS".ALARMS.WARNINGS."740170" := "DB2103_ELECTRICAL_CABINET"."0FC22_BREAKER_WARNING";
END_REGION

REGION Network 71: 0FC23 CIRCUIT BREAKER TRIPPED WARNING
   RUNG wire#powerrail
      Contact( "DB2103_ELECTRICAL_CABINET".INPUT_BREAKER_0FC23 )
      wire#w1
      Coil( "DB2103_ELECTRICAL_CABINET"."0FC23_BREAKER_WARNING" )
   END_RUNG
   RUNG wire#powerrail
      Contact( "DB2103_ELECTRICAL_CABINET"."0FC23_BREAKER_WARNING" )
      I_Contact( "DB2120_MPP_ITC_IPC".RESET_FAULTS )
   END_RUNG wire#w1
   RUNG wire#w1
      Coil( "DB426_ALARMS_WARNINGS".ALARMS.WARNINGS."740171" )
   END_RUNG
   // the same network as SCL:
   "DB2103_ELECTRICAL_CABINET"."0FC23_BREAKER_WARNING" := "DB2103_ELECTRICAL_CABINET".INPUT_BREAKER_0FC23 OR ("DB2103_ELECTRICAL_CABINET"."0FC23_BREAKER_WARNING" AND NOT "DB2120_MPP_ITC_IPC".RESET_FAULTS);
   "DB426_ALARMS_WARNINGS".ALARMS.WARNINGS."740171" := "DB2103_ELECTRICAL_CABINET"."0FC23_BREAKER_WARNING";
END_REGION

REGION Network 72: WARNINGS
   RUNG wire#powerrail
      I_Contact( "DB2103_ELECTRICAL_CABINET"."110/120/220/230VAC_BREAKER_TRIPPED_WARNING" )
      I_Contact( "DB2103_ELECTRICAL_CABINET".CAB_LIGHT_BREAKER_TRIPPED_WARNING )
      I_Contact( "DB2103_ELECTRICAL_CABINET".SENTRON_PAC_BREAKER_TRIPPED_WARNING )
      I_Contact( "DB2103_ELECTRICAL_CABINET".WATTMETER_BREAKER_TRIPPED_WARNING )
      I_Contact( "DB2103_ELECTRICAL_CABINET".ELEC_CAB_DOOR_OPEN_WARNING )
      I_Contact( "DB2103_ELECTRICAL_CABINET".BATTERY_85_SITOP_UPS500S_WARNING )
      I_Contact( "DB2103_ELECTRICAL_CABINET"."0FC20_BREAKER_WARNING" )
      I_Contact( "DB2103_ELECTRICAL_CABINET"."0FC21_BREAKER_WARNING" )
      I_Contact( "DB2103_ELECTRICAL_CABINET"."0FC22_BREAKER_WARNING" )
      I_Contact( "DB2103_ELECTRICAL_CABINET"."0FC23_BREAKER_WARNING" )
      Not()
      Coil( "DB2103_ELECTRICAL_CABINET".WARNINGS )
      { S7_GenerateENO := "TRUE" } Move(in := #FC_NUMBER, out1 => "DB440_MACHINE_ALARM_DECODING".GLOBAL_ALARMS_MACHINE.WARNING_DECODING)
      wire#w1
      S_Coil( "DB440_MACHINE_ALARM_DECODING".ALARMS_CENTRAL.WARNING )
   END_RUNG
   RUNG wire#w1
      N_Trig( "DB2103_ELECTRICAL_CABINET".WARNINGS_GONE )
      { S7_GenerateENO := "TRUE" } Move(in := 0, out1 => "DB440_MACHINE_ALARM_DECODING".GLOBAL_ALARMS_MACHINE.WARNING_DECODING)
      R_Coil( "DB440_MACHINE_ALARM_DECODING".ALARMS_CENTRAL.WARNING )
   END_RUNG
   // the same network as SCL:
   // ENO of a box is taken as its EN; it also drops when the box reports an error
   "DB2103_ELECTRICAL_CABINET".WARNINGS := NOT (NOT "DB2103_ELECTRICAL_CABINET"."110/120/220/230VAC_BREAKER_TRIPPED_WARNING" AND NOT "DB2103_ELECTRICAL_CABINET".CAB_LIGHT_BREAKER_TRIPPED_WARNING AND NOT "DB2103_ELECTRICAL_CABINET".SENTRON_PAC_BREAKER_TRIPPED_WARNING AND NOT "DB2103_ELECTRICAL_CABINET".WATTMETER_BREAKER_TRIPPED_WARNING AND NOT "DB2103_ELECTRICAL_CABINET".ELEC_CAB_DOOR_OPEN_WARNING AND NOT "DB2103_ELECTRICAL_CABINET".BATTERY_85_SITOP_UPS500S_WARNING AND NOT "DB2103_ELECTRICAL_CABINET"."0FC20_BREAKER_WARNING" AND NOT "DB2103_ELECTRICAL_CABINET"."0FC21_BREAKER_WARNING" AND NOT "DB2103_ELECTRICAL_CABINET"."0FC22_BREAKER_WARNING" AND NOT "DB2103_ELECTRICAL_CABINET"."0FC23_BREAKER_WARNING");
   IF "DB2103_ELECTRICAL_CABINET".WARNINGS THEN
       "DB440_MACHINE_ALARM_DECODING".GLOBAL_ALARMS_MACHINE.WARNING_DECODING := #FC_NUMBER;
       "DB440_MACHINE_ALARM_DECODING".ALARMS_CENTRAL.WARNING := TRUE;
   END_IF;
   #_w1 := NOT "DB2103_ELECTRICAL_CABINET".WARNINGS AND "DB2103_ELECTRICAL_CABINET".WARNINGS_GONE;   // falling edge
   "DB2103_ELECTRICAL_CABINET".WARNINGS_GONE := "DB2103_ELECTRICAL_CABINET".WARNINGS;
   IF #_w1 THEN
       "DB440_MACHINE_ALARM_DECODING".GLOBAL_ALARMS_MACHINE.WARNING_DECODING := 0;
       "DB440_MACHINE_ALARM_DECODING".ALARMS_CENTRAL.WARNING := FALSE;
   END_IF;
END_REGION
END_FUNCTION
